LIN {X 0,Y 282.516,Z 713.635,A -85,B 0,C 180,E1 -17402.793,E2 -17402.793} C_VEL
LIN {X 0,Y 282.335,Z 708.345,A -85,B 0,C 180,E1 -17403.944,E2 -17403.944} C_VEL
LIN {X 0,Y 281.852,Z 698.641,A -85,B 0,C 180,E1 -17406.313,E2 -17406.313} C_VEL
LIN {X 0,Y 281.853,Z 692.587,A -85,B 0,C 180,E1 -17407.889,E2 -17407.889} C_VEL
LIN {X 0,Y 281.9,Z 689.303,A -85,B 0,C 180,E1 -17409.389,E2 -17409.389} C_VEL
LIN {X 0,Y 280.609,Z 682.822,A -85,B 0,C 180,E1 -17412.548,E2 -17412.548} C_VEL
LIN {X 0,Y 278.888,Z 673.925,A -85,B 0,C 180,E1 -17417.125,E2 -17417.125} C_VEL
LIN {X 0,Y 277.605,Z 667.473,A -85,B 0,C 180,E1 -17420.734,E2 -17420.734} C_VEL
LIN {X 0,Y 277.296,Z 665.936,A -85,B 0,C 180,E1 -17422.76,E2 -17422.76} C_VEL
LIN {X 0,Y 277.252,Z 665.949,A -85,B 0,C 180,E1 -17426.771,E2 -17426.771} C_VEL
LIN {X 0,Y 277.258,Z 665.946,A -85,B 0,C 180,E1 -17429.538,E2 -17429.538} C_VEL
LIN {X 0,Y 277.355,Z 665.938,A -85,B 0,C 180,E1 -17432.863,E2 -17432.863} C_VEL
LIN {X 0,Y 277.346,Z 666.111,A -85,B 0,C 180,E1 -17435.612,E2 -17435.612} C_VEL
LIN {X 0,Y 278.317,Z 668.775,A -85,B 0,C 180,E1 -17439.297,E2 -17439.297} C_VEL
LIN {X 0,Y 279.682,Z 671.989,A -85,B 0,C 180,E1 -17442.72,E2 -17442.72} C_VEL
LIN {X 0,Y 280.839,Z 675.261,A -85,B 0,C 180,E1 -17445.507,E2 -17445.507} C_VEL
LIN {X 0,Y 282.859,Z 681.56,A -85,B 0,C 180,E1 -17449.984,E2 -17449.984} C_VEL
LIN {X 0,Y 284.181,Z 686.268,A -85,B 0,C 180,E1 -17452.897,E2 -17452.897} C_VEL
LIN {X 0,Y 285.808,Z 694.293,A -85,B 0,C 180,E1 -17457.181,E2 -17457.181} C_VEL
LIN {X 0,Y 286.354,Z 698.631,A -85,B 0,C 180,E1 -17459.297,E2 -17459.297} C_VEL
LIN {X 0,Y 286.469,Z 703.417,A -85,B 0,C 180,E1 -17461.406,E2 -17461.406} C_VEL
LIN {X 0,Y 285.558,Z 710.397,A -85,B 0,C 180,E1 -17464.234,E2 -17464.234} C_VEL
LIN {X 0,Y 283.691,Z 723.175,A -85,B 0,C 180,E1 -17469.266,E2 -17469.266} C_VEL
LIN {X 0,Y 282.575,Z 731.62,A -85,B 0,C 180,E1 -17472.569,E2 -17472.569} C_VEL
LIN {X 0,Y 286.588,Z 745.3,A -85,B 0,C 180,E1 -17473.876,E2 -17473.876} C_VEL
LIN {X 0,Y 288.999,Z 757.39,A -85,B 0,C 180,E1 -17475.109,E2 -17475.109} C_VEL
LIN {X 0,Y 290.187,Z 767.895,A -85,B 0,C 180,E1 -17476.293,E2 -17476.293} C_VEL
LIN {X 0,Y 290.327,Z 771.233,A -85,B 0,C 180,E1 -17476.686,E2 -17476.686} C_VEL
LIN {X 0,Y 288.563,Z 782.164,A -85,B 0,C 180,E1 -17477.917,E2 -17477.917} C_VEL
LIN {X 0,Y 286.272,Z 793.647,A -85,B 0,C 180,E1 -17479.542,E2 -17479.542} C_VEL
LIN {X 0,Y 284.389,Z 802.419,A -85,B 0,C 180,E1 -17481.084,E2 -17481.084} C_VEL
LIN {X 0,Y 282.37,Z 811.035,A -85,B 0,C 180,E1 -17482.945,E2 -17482.945} C_VEL
LIN {X 0,Y 280.37,Z 819.405,A -85,B 0,C 180,E1 -17485.222,E2 -17485.222} C_VEL
LIN {X 0,Y 278.741,Z 825.869,A -85,B 0,C 180,E1 -17487.438,E2 -17487.438} C_VEL
LIN {X 0,Y 277.545,Z 830.747,A -85,B 0,C 180,E1 -17489.571,E2 -17489.571} C_VEL
LIN {X 0,Y 276.408,Z 835.334,A -85,B 0,C 180,E1 -17492.273,E2 -17492.273} C_VEL
LIN {X 0,Y 275.833,Z 837.589,A -85,B 0,C 180,E1 -17494.093,E2 -17494.093} C_VEL
LIN {X 0,Y 275.381,Z 839.172,A -85,B 0,C 180,E1 -17495.943,E2 -17495.943} C_VEL
LIN {X 0,Y 275.105,Z 840.115,A -85,B 0,C 180,E1 -17497.815,E2 -17497.815} C_VEL
LIN {X 0,Y 274.936,Z 840.404,A -85,B 0,C 180,E1 -17499.928,E2 -17499.928} C_VEL
LIN {X 0,Y 274.846,Z 839.806,A -85,B 0,C 180,E1 -17502.138,E2 -17502.138} C_VEL
LIN {X 0,Y 274.987,Z 838.312,A -85,B 0,C 180,E1 -17504.308,E2 -17504.308} C_VEL
LIN {X 0,Y 275.3,Z 835.946,A -85,B 0,C 180,E1 -17506.429,E2 -17506.429} C_VEL
LIN {X 0,Y 275.731,Z 832.732,A -85,B 0,C 180,E1 -17508.495,E2 -17508.495} C_VEL
LIN {X 0,Y 276.231,Z 828.679,A -85,B 0,C 180,E1 -17510.503,E2 -17510.503} C_VEL
LIN {X 0,Y 277.201,Z 822.448,A -85,B 0,C 180,E1 -17512.917,E2 -17512.917} C_VEL
LIN {X 0,Y 278.175,Z 815.947,A -85,B 0,C 180,E1 -17514.911,E2 -17514.911} C_VEL
LIN {X 0,Y 279.558,Z 807.198,A -85,B 0,C 180,E1 -17517.069,E2 -17517.069} C_VEL
LIN {X 0,Y 281.061,Z 797.536,A -85,B 0,C 180,E1 -17518.985,E2 -17518.985} C_VEL
LIN {X 0,Y 282.714,Z 786.024,A -85,B 0,C 180,E1 -17520.79,E2 -17520.79} C_VEL
LIN {X 0,Y 284.124,Z 775.276,A -85,B 0,C 180,E1 -17522.131,E2 -17522.131} C_VEL
LIN {X 0,Y 285.075,Z 766.778,A -85,B 0,C 180,E1 -17522.987,E2 -17522.987} C_VEL
LIN {X 0,Y 283.775,Z 755.666,A -85,B 0,C 180,E1 -17524.046,E2 -17524.046} C_VEL
LIN {X 0,Y 281.716,Z 742.537,A -85,B 0,C 180,E1 -17525.035,E2 -17525.035} C_VEL
LIN {X 0,Y 279.529,Z 730.489,A -85,B 0,C 180,E1 -17525.738,E2 -17525.738} C_VEL
LIN {X 0,Y 280.502,Z 719.526,A -85,B 0,C 180,E1 -17529.849,E2 -17529.849} C_VEL
LIN {X 0,Y 281.518,Z 708.313,A -85,B 0,C 180,E1 -17534.062,E2 -17534.062} C_VEL
LIN {X 0,Y 282.397,Z 698.443,A -85,B 0,C 180,E1 -17537.788,E2 -17537.788} C_VEL
LIN {X 0,Y 282.636,Z 692.781,A -85,B 0,C 180,E1 -17539.977,E2 -17539.977} C_VEL
LIN {X 0,Y 281.744,Z 685.786,A -85,B 0,C 180,E1 -17542.836,E2 -17542.836} C_VEL
LIN {X 0,Y 280.07,Z 677.374,A -85,B 0,C 180,E1 -17546.404,E2 -17546.404} C_VEL
LIN {X 0,Y 278.607,Z 668.999,A -85,B 0,C 180,E1 -17550.001,E2 -17550.001} C_VEL
LIN {X 0,Y 277.825,Z 665.875,A -85,B 0,C 180,E1 -17551.45,E2 -17551.45} C_VEL
LIN {X 0,Y 277.651,Z 665.897,A -85,B 0,C 180,E1 -17557.272,E2 -17557.272} C_VEL
LIN {X 0,Y 277.508,Z 665.911,A -85,B 0,C 180,E1 -17560.212,E2 -17560.212} C_VEL
LIN {X 0,Y 277.436,Z 665.927,A -85,B 0,C 180,E1 -17564.16,E2 -17564.16} C_VEL
LIN {X 0,Y 281.89,Z 679.397,A -85,B 0,C 180,E1 -17565.735,E2 -17565.735} C_VEL
LIN {X 0,Y 284.669,Z 688.988,A -85,B 0,C 180,E1 -17567.051,E2 -17567.051} C_VEL
LIN {X 0,Y 285.979,Z 694.54,A -85,B 0,C 180,E1 -17567.891,E2 -17567.891} C_VEL
LIN {X 0,Y 284.721,Z 705.21,A -85,B 0,C 180,E1 -17569.466,E2 -17569.466} C_VEL
LIN {X 0,Y 283.372,Z 715.102,A -85,B 0,C 180,E1 -17571.268,E2 -17571.268} C_VEL
LIN {X 0,Y 282.092,Z 723.419,A -85,B 0,C 180,E1 -17573.126,E2 -17573.126} C_VEL
LIN {X 0,Y 280.89,Z 730.843,A -85,B 0,C 180,E1 -17575.173,E2 -17575.173} C_VEL
LIN {X 0,Y 279.764,Z 737.817,A -85,B 0,C 180,E1 -17577.59,E2 -17577.59} C_VEL
LIN {X 0,Y 278.868,Z 743.707,A -85,B 0,C 180,E1 -17580.268,E2 -17580.268} C_VEL
LIN {X 0,Y 278.373,Z 746.65,A -85,B 0,C 180,E1 -17582.018,E2 -17582.018} C_VEL
LIN {X 0,Y 278.006,Z 748.956,A -85,B 0,C 180,E1 -17583.791,E2 -17583.791} C_VEL
LIN {X 0,Y 277.752,Z 750.928,A -85,B 0,C 180,E1 -17585.934,E2 -17585.934} C_VEL
LIN {X 0,Y 277.767,Z 752.085,A -85,B 0,C 180,E1 -17588.339,E2 -17588.339} C_VEL
LIN {X 0,Y 278.168,Z 752.088,A -85,B 0,C 180,E1 -17591.064,E2 -17591.064} C_VEL
LIN {X 0,Y 278.594,Z 751.262,A -85,B 0,C 180,E1 -17592.982,E2 -17592.982} C_VEL
LIN {X 0,Y 279.307,Z 749.426,A -85,B 0,C 180,E1 -17595.207,E2 -17595.207} C_VEL
LIN {X 0,Y 280.569,Z 745.778,A -85,B 0,C 180,E1 -17597.935,E2 -17597.935} C_VEL
LIN {X 0,Y 282.038,Z 740.635,A -85,B 0,C 180,E1 -17600.578,E2 -17600.578} C_VEL
LIN {X 0,Y 283.861,Z 734.085,A -85,B 0,C 180,E1 -17603.052,E2 -17603.052} C_VEL
LIN {X 0,Y 285.785,Z 726.31,A -85,B 0,C 180,E1 -17605.317,E2 -17605.317} C_VEL
LIN {X 0,Y 287.637,Z 717.926,A -85,B 0,C 180,E1 -17607.249,E2 -17607.249} C_VEL
LIN {X 0,Y 289.479,Z 709.01,A -85,B 0,C 180,E1 -17608.9,E2 -17608.9} C_VEL
LIN {X 0,Y 290.619,Z 701.513,A -85,B 0,C 180,E1 -17610.082,E2 -17610.082} C_VEL
LIN {X 0,Y 288.425,Z 693.11,A -85,B 0,C 180,E1 -17611.631,E2 -17611.631} C_VEL
LIN {X 0,Y 285.145,Z 683.447,A -85,B 0,C 180,E1 -17613.269,E2 -17613.269} C_VEL
LIN {X 0,Y 280.932,Z 673.769,A -85,B 0,C 180,E1 -17614.832,E2 -17614.832} C_VEL
LIN {X 0,Y 278.336,Z 668.845,A -85,B 0,C 180,E1 -17615.621,E2 -17615.621} C_VEL
LIN {X 0,Y 277.301,Z 665.938,A -85,B 0,C 180,E1 -17616,E2 -17616} C_VEL
LIN {X 0,Y 277.347,Z 665.939,A -85,B 0,C 180,E1 -17620.767,E2 -17620.767} C_VEL
LIN {X 0,Y 277.437,Z 665.925,A -85,B 0,C 180,E1 -17625.326,E2 -17625.326} C_VEL
LIN {X 0,Y 277.406,Z 665.927,A -85,B 0,C 180,E1 -17625.963,E2 -17625.963} C_VEL
LIN {X 0,Y 276.737,Z 666.015,A -85,B 0,C 180,E1 -17627.175,E2 -17627.175} C_VEL
LIN {X 0,Y 273.935,Z 666.357,A -85,B 0,C 180,E1 -17629.153,E2 -17629.153} C_VEL
LIN {X 0,Y 271.603,Z 666.652,A -85,B 0,C 180,E1 -17630.761,E2 -17630.761} C_VEL
LIN {X 0,Y 270.654,Z 666.761,A -85,B 0,C 180,E1 -17632.004,E2 -17632.004} C_VEL
LIN {X 0,Y 270.604,Z 666.766,A -85,B 0,C 180,E1 -17632.425,E2 -17632.425} C_VEL
LIN {X 0,Y 270.79,Z 666.754,A -85,B 0,C 180,E1 -17638.513,E2 -17638.513} C_VEL
LIN {X 0,Y 270.79,Z 666.742,A -85,B 0,C 180,E1 -17641.487,E2 -17641.487} C_VEL
LIN {X 0,Y 270.614,Z 666.776,A -85,B 0,C 180,E1 -17647.461,E2 -17647.461} C_VEL
LIN {X 0,Y 270.444,Z 666.795,A -85,B 0,C 180,E1 -17650.481,E2 -17650.481} C_VEL
LIN {X 0,Y 270.406,Z 666.802,A -85,B 0,C 180,E1 -17655.065,E2 -17655.065} C_VEL
LIN {X 0,Y 270.304,Z 666.807,A -85,B 0,C 180,E1 -17659.756,E2 -17659.756} C_VEL
LIN {X 0,Y 270.276,Z 666.819,A -85,B 0,C 180,E1 -17664.586,E2 -17664.586} C_VEL
LIN {X 0,Y 270.272,Z 666.816,A -85,B 0,C 180,E1 -17667.909,E2 -17667.909} C_VEL
LIN {X 0,Y 270.187,Z 666.83,A -85,B 0,C 180,E1 -17671.348,E2 -17671.348} C_VEL
LIN {X 0,Y 270.224,Z 666.943,A -85,B 0,C 180,E1 -17673.529,E2 -17673.529} C_VEL
LIN {X 0,Y 271.355,Z 671.877,A -85,B 0,C 180,E1 -17677.492,E2 -17677.492} C_VEL
LIN {X 0,Y 272.72,Z 678.439,A -85,B 0,C 180,E1 -17682.069,E2 -17682.069} C_VEL
LIN {X 0,Y 273.966,Z 685.04,A -85,B 0,C 180,E1 -17686.161,E2 -17686.161} C_VEL
LIN {X 0,Y 275.274,Z 692.519,A -85,B 0,C 180,E1 -17690.336,E2 -17690.336} C_VEL
LIN {X 0,Y 275.316,Z 694.363,A -85,B 0,C 180,E1 -17691.287,E2 -17691.287} C_VEL
LIN {X 0,Y 273.666,Z 702.79,A -85,B 0,C 180,E1 -17695.265,E2 -17695.265} C_VEL
LIN {X 0,Y 271.808,Z 713.574,A -85,B 0,C 180,E1 -17700.149,E2 -17700.149} C_VEL
LIN {X 0,Y 271.718,Z 714.564,A -85,B 0,C 180,E1 -17700.511,E2 -17700.511} C_VEL
LIN {X 0,Y 274.842,Z 729.066,A -85,B 0,C 180,E1 -17701.706,E2 -17701.706} C_VEL
LIN {X 0,Y 276.656,Z 742.403,A -85,B 0,C 180,E1 -17702.962,E2 -17702.962} C_VEL
LIN {X 0,Y 277.427,Z 754.489,A -85,B 0,C 180,E1 -17704.276,E2 -17704.276} C_VEL
LIN {X 0,Y 277.294,Z 766.965,A -85,B 0,C 180,E1 -17705.842,E2 -17705.842} C_VEL
LIN {X 0,Y 276.639,Z 775.939,A -85,B 0,C 180,E1 -17707.11,E2 -17707.11} C_VEL
LIN {X 0,Y 276.576,Z 788.697,A -85,B 0,C 180,E1 -17708.379,E2 -17708.379} C_VEL
LIN {X 0,Y 275.815,Z 796.463,A -85,B 0,C 180,E1 -17709.295,E2 -17709.295} C_VEL
LIN {X 0,Y 274.239,Z 806.674,A -85,B 0,C 180,E1 -17710.734,E2 -17710.734} C_VEL
LIN {X 0,Y 272.809,Z 816.634,A -85,B 0,C 180,E1 -17712.483,E2 -17712.483} C_VEL
LIN {X 0,Y 271.598,Z 824.755,A -85,B 0,C 180,E1 -17714.234,E2 -17714.234} C_VEL
LIN {X 0,Y 270.302,Z 833.109,A -85,B 0,C 180,E1 -17716.466,E2 -17716.466} C_VEL
LIN {X 0,Y 269.369,Z 839.817,A -85,B 0,C 180,E1 -17718.715,E2 -17718.715} C_VEL
LIN {X 0,Y 268.762,Z 845.144,A -85,B 0,C 180,E1 -17720.972,E2 -17720.972} C_VEL
LIN {X 0,Y 268.426,Z 849.255,A -85,B 0,C 180,E1 -17723.233,E2 -17723.233} C_VEL
LIN {X 0,Y 268.262,Z 852.262,A -85,B 0,C 180,E1 -17725.491,E2 -17725.491} C_VEL
LIN {X 0,Y 268.275,Z 853.702,A -85,B 0,C 180,E1 -17726.996,E2 -17726.996} C_VEL
LIN {X 0,Y 268.277,Z 854.694,A -85,B 0,C 180,E1 -17728.498,E2 -17728.498} C_VEL
LIN {X 0,Y 268.298,Z 855.284,A -85,B 0,C 180,E1 -17729.999,E2 -17729.999} C_VEL
LIN {X 0,Y 268.265,Z 855.467,A -85,B 0,C 180,E1 -17731.5,E2 -17731.5} C_VEL
LIN {X 0,Y 268.247,Z 855.199,A -85,B 0,C 180,E1 -17733.003,E2 -17733.003} C_VEL
LIN {X 0,Y 268.31,Z 853.465,A -85,B 0,C 180,E1 -17736.013,E2 -17736.013} C_VEL
LIN {X 0,Y 268.52,Z 851.985,A -85,B 0,C 180,E1 -17737.519,E2 -17737.519} C_VEL
LIN {X 0,Y 269.047,Z 848.948,A -85,B 0,C 180,E1 -17739.775,E2 -17739.775} C_VEL
LIN {X 0,Y 269.882,Z 844.869,A -85,B 0,C 180,E1 -17742.023,E2 -17742.023} C_VEL
LIN {X 0,Y 271.316,Z 838.624,A -85,B 0,C 180,E1 -17744.628,E2 -17744.628} C_VEL
LIN {X 0,Y 273.088,Z 831.856,A -85,B 0,C 180,E1 -17746.828,E2 -17746.828} C_VEL
LIN {X 0,Y 274.777,Z 824.228,A -85,B 0,C 180,E1 -17748.851,E2 -17748.851} C_VEL
LIN {X 0,Y 276.976,Z 815.012,A -85,B 0,C 180,E1 -17750.807,E2 -17750.807} C_VEL
LIN {X 0,Y 279.372,Z 804.653,A -85,B 0,C 180,E1 -17752.558,E2 -17752.558} C_VEL
LIN {X 0,Y 281.353,Z 794.523,A -85,B 0,C 180,E1 -17753.947,E2 -17753.947} C_VEL
LIN {X 0,Y 282.205,Z 783.816,A -85,B 0,C 180,E1 -17755.237,E2 -17755.237} C_VEL
LIN {X 0,Y 282.791,Z 772.129,A -85,B 0,C 180,E1 -17756.367,E2 -17756.367} C_VEL
LIN {X 0,Y 282.217,Z 761.442,A -85,B 0,C 180,E1 -17757.306,E2 -17757.306} C_VEL
LIN {X 0,Y 280.394,Z 749.6,A -85,B 0,C 180,E1 -17758.265,E2 -17758.265} C_VEL
LIN {X 0,Y 277.549,Z 737.167,A -85,B 0,C 180,E1 -17759.29,E2 -17759.29} C_VEL
LIN {X 0,Y 276.992,Z 723.016,A -85,B 0,C 180,E1 -17761.98,E2 -17761.98} C_VEL
LIN {X 0,Y 276.498,Z 710.459,A -85,B 0,C 180,E1 -17764.762,E2 -17764.762} C_VEL
LIN {X 0,Y 276.237,Z 700.914,A -85,B 0,C 180,E1 -17767.173,E2 -17767.173} C_VEL
LIN {X 0,Y 276.348,Z 695.937,A -85,B 0,C 180,E1 -17768.539,E2 -17768.539} C_VEL
LIN {X 0,Y 275.257,Z 690.441,A -85,B 0,C 180,E1 -17770.572,E2 -17770.572} C_VEL
LIN {X 0,Y 273.681,Z 683.277,A -85,B 0,C 180,E1 -17773.894,E2 -17773.894} C_VEL
LIN {X 0,Y 272.784,Z 677.893,A -85,B 0,C 180,E1 -17776.941,E2 -17776.941} C_VEL
LIN {X 0,Y 272.529,Z 672.615,A -85,B 0,C 180,E1 -17780.68,E2 -17780.68} C_VEL
LIN {X 0,Y 272.368,Z 671.627,A -85,B 0,C 180,E1 -17781.736,E2 -17781.736} C_VEL
LIN {X 0,Y 271.899,Z 670.538,A -85,B 0,C 180,E1 -17783.523,E2 -17783.523} C_VEL
LIN {X 0,Y 271.093,Z 669.499,A -85,B 0,C 180,E1 -17787.015,E2 -17787.015} C_VEL
LIN {X 0,Y 271.016,Z 669.352,A -85,B 0,C 180,E1 -17790.481,E2 -17790.481} C_VEL
LIN {X 0,Y 271.763,Z 670.36,A -85,B 0,C 180,E1 -17794.837,E2 -17794.837} C_VEL
LIN {X 0,Y 272.599,Z 672.91,A -85,B 0,C 180,E1 -17798.842,E2 -17798.842} C_VEL
LIN {X 0,Y 273.689,Z 675.62,A -85,B 0,C 180,E1 -17802.052,E2 -17802.052} C_VEL
LIN {X 0,Y 275.21,Z 680.045,A -85,B 0,C 180,E1 -17806.02,E2 -17806.02} C_VEL
LIN {X 0,Y 276.81,Z 685.119,A -85,B 0,C 180,E1 -17809.762,E2 -17809.762} C_VEL
LIN {X 0,Y 278.052,Z 689.768,A -85,B 0,C 180,E1 -17812.739,E2 -17812.739} C_VEL
LIN {X 0,Y 279.519,Z 697.573,A -85,B 0,C 180,E1 -17817.117,E2 -17817.117} C_VEL
LIN {X 0,Y 280.009,Z 702.002,A -85,B 0,C 180,E1 -17819.281,E2 -17819.281} C_VEL
LIN {X 0,Y 279.929,Z 706.769,A -85,B 0,C 180,E1 -17821.438,E2 -17821.438} C_VEL
LIN {X 0,Y 278.841,Z 713.804,A -85,B 0,C 180,E1 -17824.336,E2 -17824.336} C_VEL
LIN {X 0,Y 277.155,Z 724.731,A -85,B 0,C 180,E1 -17828.751,E2 -17828.751} C_VEL
LIN {X 0,Y 276.136,Z 731.883,A -85,B 0,C 180,E1 -17831.608,E2 -17831.608} C_VEL
LIN {X 0,Y 280.408,Z 746.094,A -85,B 0,C 180,E1 -17833.036,E2 -17833.036} C_VEL
LIN {X 0,Y 282.806,Z 758.54,A -85,B 0,C 180,E1 -17834.389,E2 -17834.389} C_VEL
LIN {X 0,Y 284,Z 770.352,A -85,B 0,C 180,E1 -17835.796,E2 -17835.796} C_VEL
LIN {X 0,Y 283.702,Z 775.24,A -85,B 0,C 180,E1 -17836.367,E2 -17836.367} C_VEL
LIN {X 0,Y 281.675,Z 785.865,A -85,B 0,C 180,E1 -17837.659,E2 -17837.659} C_VEL
LIN {X 0,Y 279.455,Z 796.319,A -85,B 0,C 180,E1 -17839.273,E2 -17839.273} C_VEL
LIN {X 0,Y 277.085,Z 806.254,A -85,B 0,C 180,E1 -17841.188,E2 -17841.188} C_VEL
LIN {X 0,Y 275.074,Z 814.242,A -85,B 0,C 180,E1 -17843.109,E2 -17843.109} C_VEL
LIN {X 0,Y 273.2,Z 821.576,A -85,B 0,C 180,E1 -17845.31,E2 -17845.31} C_VEL
LIN {X 0,Y 271.388,Z 828.098,A -85,B 0,C 180,E1 -17847.784,E2 -17847.784} C_VEL
LIN {X 0,Y 270.164,Z 832.914,A -85,B 0,C 180,E1 -17850.18,E2 -17850.18} C_VEL
LIN {X 0,Y 269.297,Z 836.161,A -85,B 0,C 180,E1 -17852.344,E2 -17852.344} C_VEL
LIN {X 0,Y 268.466,Z 839.02,A -85,B 0,C 180,E1 -17855.164,E2 -17855.164} C_VEL
LIN {X 0,Y 267.967,Z 840.473,A -85,B 0,C 180,E1 -17858.113,E2 -17858.113} C_VEL
LIN {X 0,Y 267.783,Z 840.39,A -85,B 0,C 180,E1 -17861.005,E2 -17861.005} C_VEL
LIN {X 0,Y 267.795,Z 839.456,A -85,B 0,C 180,E1 -17863.027,E2 -17863.027} C_VEL
LIN {X 0,Y 268.136,Z 836.58,A -85,B 0,C 180,E1 -17866.077,E2 -17866.077} C_VEL
LIN {X 0,Y 268.571,Z 833.554,A -85,B 0,C 180,E1 -17868.182,E2 -17868.182} C_VEL
LIN {X 0,Y 269.219,Z 828.568,A -85,B 0,C 180,E1 -17870.756,E2 -17870.756} C_VEL
LIN {X 0,Y 270.232,Z 822.128,A -85,B 0,C 180,E1 -17873.263,E2 -17873.263} C_VEL
LIN {X 0,Y 271.452,Z 814.368,A -85,B 0,C 180,E1 -17875.622,E2 -17875.622} C_VEL
LIN {X 0,Y 272.882,Z 805.731,A -85,B 0,C 180,E1 -17877.718,E2 -17877.718} C_VEL
LIN {X 0,Y 274.556,Z 795.036,A -85,B 0,C 180,E1 -17879.778,E2 -17879.778} C_VEL
LIN {X 0,Y 276.174,Z 784.204,A -85,B 0,C 180,E1 -17881.437,E2 -17881.437} C_VEL
LIN {X 0,Y 277.521,Z 773.78,A -85,B 0,C 180,E1 -17882.71,E2 -17882.71} C_VEL
LIN {X 0,Y 278.159,Z 766.612,A -85,B 0,C 180,E1 -17883.45,E2 -17883.45} C_VEL
LIN {X 0,Y 276.72,Z 754.813,A -85,B 0,C 180,E1 -17884.596,E2 -17884.596} C_VEL
LIN {X 0,Y 274.596,Z 741.045,A -85,B 0,C 180,E1 -17885.63,E2 -17885.63} C_VEL
LIN {X 0,Y 272.611,Z 730.637,A -85,B 0,C 180,E1 -17886.247,E2 -17886.247} C_VEL
LIN {X 0,Y 273.6,Z 720.504,A -85,B 0,C 180,E1 -17890.103,E2 -17890.103} C_VEL
LIN {X 0,Y 274.655,Z 709.243,A -85,B 0,C 180,E1 -17894.415,E2 -17894.415} C_VEL
LIN {X 0,Y 275.579,Z 699.289,A -85,B 0,C 180,E1 -17898.229,E2 -17898.229} C_VEL
LIN {X 0,Y 275.72,Z 693.635,A -85,B 0,C 180,E1 -17900.464,E2 -17900.464} C_VEL
LIN {X 0,Y 274.774,Z 686.612,A -85,B 0,C 180,E1 -17903.392,E2 -17903.392} C_VEL
LIN {X 0,Y 272.555,Z 674.785,A -85,B 0,C 180,E1 -17908.523,E2 -17908.523} C_VEL
LIN {X 0,Y 271.508,Z 669.803,A -85,B 0,C 180,E1 -17910.742,E2 -17910.742} C_VEL
LIN {X 0,Y 270.71,Z 666.763,A -85,B 0,C 180,E1 -17912.233,E2 -17912.233} C_VEL
LIN {X 0,Y 270.609,Z 666.775,A -85,B 0,C 180,E1 -17917.462,E2 -17917.462} C_VEL
LIN {X 0,Y 270.443,Z 666.793,A -85,B 0,C 180,E1 -17920.482,E2 -17920.482} C_VEL
LIN {X 0,Y 270.406,Z 666.804,A -85,B 0,C 180,E1 -17923.624,E2 -17923.624} C_VEL
LIN {X 0,Y 274.776,Z 679.978,A -85,B 0,C 180,E1 -17925.199,E2 -17925.199} C_VEL
LIN {X 0,Y 277.625,Z 689.557,A -85,B 0,C 180,E1 -17926.547,E2 -17926.547} C_VEL
LIN {X 0,Y 279.157,Z 696.219,A -85,B 0,C 180,E1 -17927.585,E2 -17927.585} C_VEL
LIN {X 0,Y 277.848,Z 706.788,A -85,B 0,C 180,E1 -17929.198,E2 -17929.198} C_VEL
LIN {X 0,Y 276.591,Z 715.581,A -85,B 0,C 180,E1 -17930.839,E2 -17930.839} C_VEL
LIN {X 0,Y 275.239,Z 724.199,A -85,B 0,C 180,E1 -17932.793,E2 -17932.793} C_VEL
LIN {X 0,Y 273.897,Z 732.171,A -85,B 0,C 180,E1 -17935.049,E2 -17935.049} C_VEL
LIN {X 0,Y 272.715,Z 739.374,A -85,B 0,C 180,E1 -17937.638,E2 -17937.638} C_VEL
LIN {X 0,Y 271.841,Z 744.913,A -85,B 0,C 180,E1 -17940.275,E2 -17940.275} C_VEL
LIN {X 0,Y 271.139,Z 749.043,A -85,B 0,C 180,E1 -17942.979,E2 -17942.979} C_VEL
LIN {X 0,Y 270.837,Z 751.025,A -85,B 0,C 180,E1 -17944.812,E2 -17944.812} C_VEL
LIN {X 0,Y 270.721,Z 752.399,A -85,B 0,C 180,E1 -17946.662,E2 -17946.662} C_VEL
LIN {X 0,Y 270.799,Z 753.217,A -85,B 0,C 180,E1 -17948.869,E2 -17948.869} C_VEL
LIN {X 0,Y 271.185,Z 753.134,A -85,B 0,C 180,E1 -17951.275,E2 -17951.275} C_VEL
LIN {X 0,Y 271.982,Z 751.621,A -85,B 0,C 180,E1 -17954.242,E2 -17954.242} C_VEL
LIN {X 0,Y 273.179,Z 748.538,A -85,B 0,C 180,E1 -17957.143,E2 -17957.143} C_VEL
LIN {X 0,Y 274.2,Z 745.441,A -85,B 0,C 180,E1 -17959.123,E2 -17959.123} C_VEL
LIN {X 0,Y 275.78,Z 740.327,A -85,B 0,C 180,E1 -17961.595,E2 -17961.595} C_VEL
LIN {X 0,Y 277.297,Z 734.91,A -85,B 0,C 180,E1 -17963.62,E2 -17963.62} C_VEL
LIN {X 0,Y 279.062,Z 728.248,A -85,B 0,C 180,E1 -17965.625,E2 -17965.625} C_VEL
LIN {X 0,Y 281.006,Z 719.94,A -85,B 0,C 180,E1 -17967.633,E2 -17967.633} C_VEL
LIN {X 0,Y 283.014,Z 710.786,A -85,B 0,C 180,E1 -17969.399,E2 -17969.399} C_VEL
LIN {X 0,Y 284.218,Z 703.649,A -85,B 0,C 180,E1 -17970.569,E2 -17970.569} C_VEL
LIN {X 0,Y 282.124,Z 695.459,A -85,B 0,C 180,E1 -17972.155,E2 -17972.155} C_VEL
LIN {X 0,Y 278.989,Z 686.089,A -85,B 0,C 180,E1 -17973.843,E2 -17973.843} C_VEL
LIN {X 0,Y 274.729,Z 676.384,A -85,B 0,C 180,E1 -17975.522,E2 -17975.522} C_VEL
LIN {X 0,Y 271.46,Z 669.995,A -85,B 0,C 180,E1 -17976.594,E2 -17976.594} C_VEL
LIN {X 0,Y 270.292,Z 667.295,A -85,B 0,C 180,E1 -17976.994,E2 -17976.994} C_VEL
LIN {X 0,Y 270.234,Z 666.811,A -85,B 0,C 180,E1 -17977.09,E2 -17977.09} C_VEL
LIN {X 0,Y 270.303,Z 666.816,A -85,B 0,C 180,E1 -17980.245,E2 -17980.245} C_VEL
LIN {X 0,Y 270.405,Z 666.804,A -85,B 0,C 180,E1 -17984.936,E2 -17984.936} C_VEL
LIN {X 0,Y 270.444,Z 666.793,A -85,B 0,C 180,E1 -17989.519,E2 -17989.519} C_VEL
LIN {X 0,Y 270.604,Z 666.766,A -85,B 0,C 180,E1 -17992.425,E2 -17992.425} C_VEL
LIN {X 0,Y 270.018,Z 666.846,A -85,B 0,C 180,E1 -17993.666,E2 -17993.666} C_VEL
LIN {X 0,Y 267.236,Z 667.195,A -85,B 0,C 180,E1 -17995.69,E2 -17995.69} C_VEL
LIN {X 0,Y 264.841,Z 667.496,A -85,B 0,C 180,E1 -17997.335,E2 -17997.335} C_VEL
LIN {X 0,Y 263.825,Z 667.621,A -85,B 0,C 180,E1 -17998.61,E2 -17998.61} C_VEL
LIN {X 0,Y 263.751,Z 667.625,A -85,B 0,C 180,E1 -17999.041,E2 -17999.041} C_VEL
LIN {X 0,Y 263.754,Z 667.619,A -85,B 0,C 180,E1 -18001.527,E2 -18001.527} C_VEL
LIN {X 0,Y 263.575,Z 667.652,A -85,B 0,C 180,E1 -18007.662,E2 -18007.662} C_VEL
LIN {X 0,Y 263.377,Z 667.679,A -85,B 0,C 180,E1 -18010.766,E2 -18010.766} C_VEL
LIN {X 0,Y 263.354,Z 667.679,A -85,B 0,C 180,E1 -18015.478,E2 -18015.478} C_VEL
LIN {X 0,Y 263.266,Z 667.684,A -85,B 0,C 180,E1 -18020.307,E2 -18020.307} C_VEL
LIN {X 0,Y 263.21,Z 667.695,A -85,B 0,C 180,E1 -18025.291,E2 -18025.291} C_VEL
LIN {X 0,Y 263.178,Z 667.7,A -85,B 0,C 180,E1 -18028.73,E2 -18028.73} C_VEL
LIN {X 0,Y 263.135,Z 667.799,A -85,B 0,C 180,E1 -18032.288,E2 -18032.288} C_VEL
LIN {X 0,Y 264.117,Z 671.885,A -85,B 0,C 180,E1 -18035.832,E2 -18035.832} C_VEL
LIN {X 0,Y 265.195,Z 677.091,A -85,B 0,C 180,E1 -18039.777,E2 -18039.777} C_VEL
LIN {X 0,Y 266.263,Z 682.303,A -85,B 0,C 180,E1 -18043.336,E2 -18043.336} C_VEL
LIN {X 0,Y 267.445,Z 688.889,A -85,B 0,C 180,E1 -18047.375,E2 -18047.375} C_VEL
LIN {X 0,Y 268.347,Z 694.049,A -85,B 0,C 180,E1 -18050.288,E2 -18050.288} C_VEL
LIN {X 0,Y 268.092,Z 697.076,A -85,B 0,C 180,E1 -18051.855,E2 -18051.855} C_VEL
LIN {X 0,Y 266.473,Z 704.694,A -85,B 0,C 180,E1 -18055.527,E2 -18055.527} C_VEL
LIN {X 0,Y 264.967,Z 713.004,A -85,B 0,C 180,E1 -18059.407,E2 -18059.407} C_VEL
LIN {X 0,Y 265.915,Z 717.051,A -85,B 0,C 180,E1 -18059.759,E2 -18059.759} C_VEL
LIN {X 0,Y 268.598,Z 730.061,A -85,B 0,C 180,E1 -18060.947,E2 -18060.947} C_VEL
LIN {X 0,Y 270.275,Z 743.125,A -85,B 0,C 180,E1 -18062.272,E2 -18062.272} C_VEL
LIN {X 0,Y 270.94,Z 754.77,A -85,B 0,C 180,E1 -18063.615,E2 -18063.615} C_VEL
LIN {X 0,Y 270.739,Z 766.246,A -85,B 0,C 180,E1 -18065.127,E2 -18065.127} C_VEL
LIN {X 0,Y 269.781,Z 777.533,A -85,B 0,C 180,E1 -18066.811,E2 -18066.811} C_VEL
LIN {X 0,Y 269.708,Z 788.94,A -85,B 0,C 180,E1 -18068.001,E2 -18068.001} C_VEL
LIN {X 0,Y 268.936,Z 796.627,A -85,B 0,C 180,E1 -18068.941,E2 -18068.941} C_VEL
LIN {X 0,Y 267.319,Z 806.772,A -85,B 0,C 180,E1 -18070.414,E2 -18070.414} C_VEL
LIN {X 0,Y 265.833,Z 816.802,A -85,B 0,C 180,E1 -18072.232,E2 -18072.232} C_VEL
LIN {X 0,Y 264.453,Z 825.502,A -85,B 0,C 180,E1 -18074.192,E2 -18074.192} C_VEL
LIN {X 0,Y 263.145,Z 833.683,A -85,B 0,C 180,E1 -18076.485,E2 -18076.485} C_VEL
LIN {X 0,Y 262.364,Z 839.241,A -85,B 0,C 180,E1 -18078.409,E2 -18078.409} C_VEL
LIN {X 0,Y 261.726,Z 844.645,A -85,B 0,C 180,E1 -18080.728,E2 -18080.728} C_VEL
LIN {X 0,Y 261.353,Z 848.825,A -85,B 0,C 180,E1 -18083.049,E2 -18083.049} C_VEL
LIN {X 0,Y 261.18,Z 851.897,A -85,B 0,C 180,E1 -18085.369,E2 -18085.369} C_VEL
LIN {X 0,Y 261.185,Z 853.396,A -85,B 0,C 180,E1 -18086.914,E2 -18086.914} C_VEL
LIN {X 0,Y 261.201,Z 854.42,A -85,B 0,C 180,E1 -18088.457,E2 -18088.457} C_VEL
LIN {X 0,Y 261.22,Z 855.038,A -85,B 0,C 180,E1 -18089.999,E2 -18089.999} C_VEL
LIN {X 0,Y 261.19,Z 855.255,A -85,B 0,C 180,E1 -18091.541,E2 -18091.541} C_VEL
LIN {X 0,Y 261.158,Z 855.04,A -85,B 0,C 180,E1 -18093.084,E2 -18093.084} C_VEL
LIN {X 0,Y 261.237,Z 853.374,A -85,B 0,C 180,E1 -18096.177,E2 -18096.177} C_VEL
LIN {X 0,Y 261.449,Z 851.948,A -85,B 0,C 180,E1 -18097.723,E2 -18097.723} C_VEL
LIN {X 0,Y 262.034,Z 848.97,A -85,B 0,C 180,E1 -18100.039,E2 -18100.039} C_VEL
LIN {X 0,Y 262.92,Z 844.964,A -85,B 0,C 180,E1 -18102.347,E2 -18102.347} C_VEL
LIN {X 0,Y 264.161,Z 839.821,A -85,B 0,C 180,E1 -18104.639,E2 -18104.639} C_VEL
LIN {X 0,Y 265.991,Z 833.393,A -85,B 0,C 180,E1 -18106.895,E2 -18106.895} C_VEL
LIN {X 0,Y 267.949,Z 825.162,A -85,B 0,C 180,E1 -18109.223,E2 -18109.223} C_VEL
LIN {X 0,Y 270.399,Z 815.678,A -85,B 0,C 180,E1 -18111.337,E2 -18111.337} C_VEL
LIN {X 0,Y 272.886,Z 805.489,A -85,B 0,C 180,E1 -18113.125,E2 -18113.125} C_VEL
LIN {X 0,Y 274.957,Z 795.57,A -85,B 0,C 180,E1 -18114.541,E2 -18114.541} C_VEL
LIN {X 0,Y 275.959,Z 785.051,A -85,B 0,C 180,E1 -18115.875,E2 -18115.875} C_VEL
LIN {X 0,Y 276.717,Z 774.001,A -85,B 0,C 180,E1 -18117.018,E2 -18117.018} C_VEL
LIN {X 0,Y 276.373,Z 763.886,A -85,B 0,C 180,E1 -18117.964,E2 -18117.964} C_VEL
LIN {X 0,Y 274.755,Z 752.009,A -85,B 0,C 180,E1 -18118.997,E2 -18118.997} C_VEL
LIN {X 0,Y 271.405,Z 737.257,A -85,B 0,C 180,E1 -18120.273,E2 -18120.273} C_VEL
LIN {X 0,Y 271.013,Z 723.771,A -85,B 0,C 180,E1 -18122.995,E2 -18122.995} C_VEL
LIN {X 0,Y 270.813,Z 714.062,A -85,B 0,C 180,E1 -18125.228,E2 -18125.228} C_VEL
LIN {X 0,Y 270.671,Z 704.472,A -85,B 0,C 180,E1 -18127.715,E2 -18127.715} C_VEL
LIN {X 0,Y 270.919,Z 700.327,A -85,B 0,C 180,E1 -18128.9,E2 -18128.9} C_VEL
LIN {X 0,Y 270.119,Z 695.671,A -85,B 0,C 180,E1 -18130.574,E2 -18130.574} C_VEL
LIN {X 0,Y 268.642,Z 688.778,A -85,B 0,C 180,E1 -18133.741,E2 -18133.741} C_VEL
LIN {X 0,Y 267.652,Z 683.02,A -85,B 0,C 180,E1 -18136.944,E2 -18136.944} C_VEL
LIN {X 0,Y 267.453,Z 677.449,A -85,B 0,C 180,E1 -18140.901,E2 -18140.901} C_VEL
LIN {X 0,Y 267.036,Z 675.931,A -85,B 0,C 180,E1 -18142.747,E2 -18142.747} C_VEL
LIN {X 0,Y 266.047,Z 674.533,A -85,B 0,C 180,E1 -18146.307,E2 -18146.307} C_VEL
LIN {X 0,Y 265.77,Z 674.123,A -85,B 0,C 180,E1 -18150.765,E2 -18150.765} C_VEL
LIN {X 0,Y 266.4,Z 675.06,A -85,B 0,C 180,E1 -18155.032,E2 -18155.032} C_VEL
LIN {X 0,Y 267.398,Z 678.216,A -85,B 0,C 180,E1 -18160.021,E2 -18160.021} C_VEL
LIN {X 0,Y 268.435,Z 681.088,A -85,B 0,C 180,E1 -18163.262,E2 -18163.262} C_VEL
LIN {X 0,Y 269.538,Z 684.62,A -85,B 0,C 180,E1 -18166.428,E2 -18166.428} C_VEL
LIN {X 0,Y 271.043,Z 689.584,A -85,B 0,C 180,E1 -18170.162,E2 -18170.162} C_VEL
LIN {X 0,Y 271.909,Z 693.229,A -85,B 0,C 180,E1 -18172.574,E2 -18172.574} C_VEL
LIN {X 0,Y 273.299,Z 701.024,A -85,B 0,C 180,E1 -18177.052,E2 -18177.052} C_VEL
LIN {X 0,Y 273.697,Z 706.906,A -85,B 0,C 180,E1 -18180,E2 -18180} C_VEL
LIN {X 0,Y 273.151,Z 711.922,A -85,B 0,C 180,E1 -18182.212,E2 -18182.212} C_VEL
LIN {X 0,Y 271.237,Z 722.701,A -85,B 0,C 180,E1 -18186.696,E2 -18186.696} C_VEL
LIN {X 0,Y 269.806,Z 732.132,A -85,B 0,C 180,E1 -18190.553,E2 -18190.553} C_VEL
LIN {X 0,Y 273.847,Z 745.446,A -85,B 0,C 180,E1 -18191.988,E2 -18191.988} C_VEL
LIN {X 0,Y 276.198,Z 756.508,A -85,B 0,C 180,E1 -18193.239,E2 -18193.239} C_VEL
LIN {X 0,Y 277.602,Z 768.151,A -85,B 0,C 180,E1 -18194.665,E2 -18194.665} C_VEL
LIN {X 0,Y 277.773,Z 774.427,A -85,B 0,C 180,E1 -18195.481,E2 -18195.481} C_VEL
LIN {X 0,Y 275.608,Z 785.625,A -85,B 0,C 180,E1 -18196.862,E2 -18196.862} C_VEL
LIN {X 0,Y 273.362,Z 795.783,A -85,B 0,C 180,E1 -18198.433,E2 -18198.433} C_VEL
LIN {X 0,Y 271.104,Z 804.857,A -85,B 0,C 180,E1 -18200.172,E2 -18200.172} C_VEL
LIN {X 0,Y 268.769,Z 813.709,A -85,B 0,C 180,E1 -18202.281,E2 -18202.281} C_VEL
LIN {X 0,Y 266.705,Z 821.184,A -85,B 0,C 180,E1 -18204.521,E2 -18204.521} C_VEL
LIN {X 0,Y 264.933,Z 827.228,A -85,B 0,C 180,E1 -18206.806,E2 -18206.806} C_VEL
LIN {X 0,Y 263.353,Z 832.857,A -85,B 0,C 180,E1 -18209.584,E2 -18209.584} C_VEL
LIN {X 0,Y 262.177,Z 836.929,A -85,B 0,C 180,E1 -18212.42,E2 -18212.42} C_VEL
LIN {X 0,Y 261.591,Z 838.852,A -85,B 0,C 180,E1 -18214.346,E2 -18214.346} C_VEL
LIN {X 0,Y 261.136,Z 840.117,A -85,B 0,C 180,E1 -18216.305,E2 -18216.305} C_VEL
LIN {X 0,Y 260.831,Z 840.792,A -85,B 0,C 180,E1 -18218.613,E2 -18218.613} C_VEL
LIN {X 0,Y 260.686,Z 840.55,A -85,B 0,C 180,E1 -18220.988,E2 -18220.988} C_VEL
LIN {X 0,Y 260.711,Z 839.404,A -85,B 0,C 180,E1 -18223.296,E2 -18223.296} C_VEL
LIN {X 0,Y 260.957,Z 837.388,A -85,B 0,C 180,E1 -18225.557,E2 -18225.557} C_VEL
LIN {X 0,Y 261.385,Z 834.513,A -85,B 0,C 180,E1 -18227.765,E2 -18227.765} C_VEL
LIN {X 0,Y 262.026,Z 829.545,A -85,B 0,C 180,E1 -18230.507,E2 -18230.507} C_VEL
LIN {X 0,Y 262.865,Z 824.396,A -85,B 0,C 180,E1 -18232.688,E2 -18232.688} C_VEL
LIN {X 0,Y 264.105,Z 816.747,A -85,B 0,C 180,E1 -18235.251,E2 -18235.251} C_VEL
LIN {X 0,Y 265.536,Z 808.333,A -85,B 0,C 180,E1 -18237.459,E2 -18237.459} C_VEL
LIN {X 0,Y 267.211,Z 798.256,A -85,B 0,C 180,E1 -18239.584,E2 -18239.584} C_VEL
LIN {X 0,Y 268.75,Z 788.148,A -85,B 0,C 180,E1 -18241.282,E2 -18241.282} C_VEL
LIN {X 0,Y 270.33,Z 776.866,A -85,B 0,C 180,E1 -18242.8,E2 -18242.8} C_VEL
LIN {X 0,Y 271.383,Z 768.818,A -85,B 0,C 180,E1 -18243.675,E2 -18243.675} C_VEL
LIN {X 0,Y 270.234,Z 758.034,A -85,B 0,C 180,E1 -18244.796,E2 -18244.796} C_VEL
LIN {X 0,Y 268.326,Z 744.948,A -85,B 0,C 180,E1 -18245.895,E2 -18245.895} C_VEL
LIN {X 0,Y 265.74,Z 730.76,A -85,B 0,C 180,E1 -18246.793,E2 -18246.793} C_VEL
LIN {X 0,Y 266.686,Z 721.477,A -85,B 0,C 180,E1 -18250.368,E2 -18250.368} C_VEL
LIN {X 0,Y 267.789,Z 710.142,A -85,B 0,C 180,E1 -18254.786,E2 -18254.786} C_VEL
LIN {X 0,Y 268.769,Z 700.139,A -85,B 0,C 180,E1 -18258.691,E2 -18258.691} C_VEL
LIN {X 0,Y 268.925,Z 696.307,A -85,B 0,C 180,E1 -18260.221,E2 -18260.221} C_VEL
LIN {X 0,Y 268.07,Z 689.203,A -85,B 0,C 180,E1 -18263.226,E2 -18263.226} C_VEL
LIN {X 0,Y 266.137,Z 678.968,A -85,B 0,C 180,E1 -18267.731,E2 -18267.731} C_VEL
LIN {X 0,Y 264.857,Z 672.26,A -85,B 0,C 180,E1 -18270.761,E2 -18270.761} C_VEL
LIN {X 0,Y 263.59,Z 667.651,A -85,B 0,C 180,E1 -18272.962,E2 -18272.962} C_VEL
LIN {X 0,Y 263.571,Z 667.653,A -85,B 0,C 180,E1 -18277.662,E2 -18277.662} C_VEL
LIN {X 0,Y 263.376,Z 667.675,A -85,B 0,C 180,E1 -18280.766,E2 -18280.766} C_VEL
LIN {X 0,Y 263.321,Z 667.687,A -85,B 0,C 180,E1 -18283.064,E2 -18283.064} C_VEL
LIN {X 0,Y 267.262,Z 679.189,A -85,B 0,C 180,E1 -18284.467,E2 -18284.467} C_VEL
LIN {X 0,Y 270.498,Z 689.858,A -85,B 0,C 180,E1 -18285.988,E2 -18285.988} C_VEL
LIN {X 0,Y 272.248,Z 696.742,A -85,B 0,C 180,E1 -18287.086,E2 -18287.086} C_VEL
LIN {X 0,Y 271.831,Z 701.91,A -85,B 0,C 180,E1 -18287.861,E2 -18287.861} C_VEL
LIN {X 0,Y 270.282,Z 712.896,A -85,B 0,C 180,E1 -18289.758,E2 -18289.758} C_VEL
LIN {X 0,Y 269.071,Z 720.859,A -85,B 0,C 180,E1 -18291.45,E2 -18291.45} C_VEL
LIN {X 0,Y 267.632,Z 729.101,A -85,B 0,C 180,E1 -18293.566,E2 -18293.566} C_VEL
LIN {X 0,Y 266.612,Z 735.353,A -85,B 0,C 180,E1 -18295.547,E2 -18295.547} C_VEL
LIN {X 0,Y 265.678,Z 740.632,A -85,B 0,C 180,E1 -18297.577,E2 -18297.577} C_VEL
LIN {X 0,Y 264.787,Z 746.106,A -85,B 0,C 180,E1 -18300.286,E2 -18300.286} C_VEL
LIN {X 0,Y 264.073,Z 750.203,A -85,B 0,C 180,E1 -18303.065,E2 -18303.065} C_VEL
LIN {X 0,Y 263.714,Z 752.906,A -85,B 0,C 180,E1 -18305.896,E2 -18305.896} C_VEL
LIN {X 0,Y 263.699,Z 753.93,A -85,B 0,C 180,E1 -18307.806,E2 -18307.806} C_VEL
LIN {X 0,Y 263.903,Z 754.344,A -85,B 0,C 180,E1 -18309.729,E2 -18309.729} C_VEL
LIN {X 0,Y 264.304,Z 754.095,A -85,B 0,C 180,E1 -18311.881,E2 -18311.881} C_VEL
LIN {X 0,Y 264.978,Z 752.884,A -85,B 0,C 180,E1 -18314.265,E2 -18314.265} C_VEL
LIN {X 0,Y 265.878,Z 750.741,A -85,B 0,C 180,E1 -18316.586,E2 -18316.586} C_VEL
LIN {X 0,Y 267.047,Z 747.643,A -85,B 0,C 180,E1 -18318.857,E2 -18318.857} C_VEL
LIN {X 0,Y 268.358,Z 743.632,A -85,B 0,C 180,E1 -18321.058,E2 -18321.058} C_VEL
LIN {X 0,Y 270.359,Z 737.238,A -85,B 0,C 180,E1 -18323.693,E2 -18323.693} C_VEL
LIN {X 0,Y 272.549,Z 729.498,A -85,B 0,C 180,E1 -18326.142,E2 -18326.142} C_VEL
LIN {X 0,Y 274.591,Z 721.267,A -85,B 0,C 180,E1 -18328.186,E2 -18328.186} C_VEL
LIN {X 0,Y 276.931,Z 711.01,A -85,B 0,C 180,E1 -18330.195,E2 -18330.195} C_VEL
LIN {X 0,Y 277.833,Z 706.45,A -85,B 0,C 180,E1 -18330.951,E2 -18330.951} C_VEL
LIN {X 0,Y 275.853,Z 697.824,A -85,B 0,C 180,E1 -18332.704,E2 -18332.704} C_VEL
LIN {X 0,Y 272.997,Z 689.08,A -85,B 0,C 180,E1 -18334.379,E2 -18334.379} C_VEL
LIN {X 0,Y 268.69,Z 678.97,A -85,B 0,C 180,E1 -18336.236,E2 -18336.236} C_VEL
LIN {X 0,Y 264.603,Z 671.132,A -85,B 0,C 180,E1 -18337.657,E2 -18337.657} C_VEL
LIN {X 0,Y 263.299,Z 668.406,A -85,B 0,C 180,E1 -18338.101,E2 -18338.101} C_VEL
LIN {X 0,Y 263.171,Z 667.697,A -85,B 0,C 180,E1 -18338.222,E2 -18338.222} C_VEL
LIN {X 0,Y 263.252,Z 667.697,A -85,B 0,C 180,E1 -18341.315,E2 -18341.315} C_VEL
LIN {X 0,Y 263.353,Z 667.684,A -85,B 0,C 180,E1 -18344.522,E2 -18344.522} C_VEL
LIN {X 0,Y 263.376,Z 667.672,A -85,B 0,C 180,E1 -18349.235,E2 -18349.235} C_VEL
LIN {X 0,Y 263.57,Z 667.642,A -85,B 0,C 180,E1 -18352.394,E2 -18352.394} C_VEL
LIN {X 0,Y 263.754,Z 667.63,A -85,B 0,C 180,E1 -18358.473,E2 -18358.473} C_VEL
LIN {X 0,Y 263.751,Z 667.625,A -85,B 0,C 180,E1 -18359.041,E2 -18359.041} C_VEL
LIN {X 0,Y 263.428,Z 667.663,A -85,B 0,C 180,E1 -18359.893,E2 -18359.893} C_VEL
LIN {X 0,Y 262.001,Z 667.842,A -85,B 0,C 180,E1 -18361.148,E2 -18361.148} C_VEL
LIN {X 0,Y 257.475,Z 668.404,A -85,B 0,C 180,E1 -18364.068,E2 -18364.068} C_VEL
LIN {X 0,Y 256.465,Z 668.526,A -85,B 0,C 180,E1 -18365.379,E2 -18365.379} C_VEL
LIN {X 0,Y 256.426,Z 668.533,A -85,B 0,C 180,E1 -18365.823,E2 -18365.823} C_VEL
LIN {X 0,Y 256.543,Z 668.525,A -85,B 0,C 180,E1 -18367.873,E2 -18367.873} C_VEL
LIN {X 0,Y 256.313,Z 668.558,A -85,B 0,C 180,E1 -18371.066,E2 -18371.066} C_VEL
LIN {X 0,Y 256.303,Z 668.552,A -85,B 0,C 180,E1 -18375.915,E2 -18375.915} C_VEL
LIN {X 0,Y 256.17,Z 668.571,A -85,B 0,C 180,E1 -18380.895,E2 -18380.895} C_VEL
LIN {X 0,Y 256.191,Z 668.57,A -85,B 0,C 180,E1 -18385.138,E2 -18385.138} C_VEL
LIN {X 0,Y 256.113,Z 668.584,A -85,B 0,C 180,E1 -18389.6,E2 -18389.6} C_VEL
LIN {X 0,Y 256.116,Z 668.669,A -85,B 0,C 180,E1 -18390.965,E2 -18390.965} C_VEL
LIN {X 0,Y 257.114,Z 673.07,A -85,B 0,C 180,E1 -18395.031,E2 -18395.031} C_VEL
LIN {X 0,Y 258.119,Z 677.767,A -85,B 0,C 180,E1 -18398.774,E2 -18398.774} C_VEL
LIN {X 0,Y 259.319,Z 683.648,A -85,B 0,C 180,E1 -18402.966,E2 -18402.966} C_VEL
LIN {X 0,Y 260.424,Z 689.622,A -85,B 0,C 180,E1 -18406.773,E2 -18406.773} C_VEL
LIN {X 0,Y 261.295,Z 694.723,A -85,B 0,C 180,E1 -18409.794,E2 -18409.794} C_VEL
LIN {X 0,Y 261.3,Z 697.44,A -85,B 0,C 180,E1 -18411.26,E2 -18411.26} C_VEL
LIN {X 0,Y 259.51,Z 705.627,A -85,B 0,C 180,E1 -18415.338,E2 -18415.338} C_VEL
LIN {X 0,Y 258.309,Z 711.807,A -85,B 0,C 180,E1 -18418.301,E2 -18418.301} C_VEL
LIN {X 0,Y 259.226,Z 715.743,A -85,B 0,C 180,E1 -18418.638,E2 -18418.638} C_VEL
LIN {X 0,Y 262.039,Z 728.793,A -85,B 0,C 180,E1 -18419.914,E2 -18419.914} C_VEL
LIN {X 0,Y 263.696,Z 740.974,A -85,B 0,C 180,E1 -18421.223,E2 -18421.223} C_VEL
LIN {X 0,Y 264.422,Z 753.313,A -85,B 0,C 180,E1 -18422.691,E2 -18422.691} C_VEL
LIN {X 0,Y 264.278,Z 764.335,A -85,B 0,C 180,E1 -18424.184,E2 -18424.184} C_VEL
LIN {X 0,Y 263.493,Z 774.16,A -85,B 0,C 180,E1 -18425.711,E2 -18425.711} C_VEL
LIN {X 0,Y 262.966,Z 778.792,A -85,B 0,C 180,E1 -18426.47,E2 -18426.47} C_VEL
LIN {X 0,Y 262.801,Z 790.833,A -85,B 0,C 180,E1 -18427.806,E2 -18427.806} C_VEL
LIN {X 0,Y 261.376,Z 800.812,A -85,B 0,C 180,E1 -18429.128,E2 -18429.128} C_VEL
LIN {X 0,Y 259.783,Z 811.236,A -85,B 0,C 180,E1 -18430.851,E2 -18430.851} C_VEL
LIN {X 0,Y 258.423,Z 819.807,A -85,B 0,C 180,E1 -18432.593,E2 -18432.593} C_VEL
LIN {X 0,Y 257.094,Z 827.709,A -85,B 0,C 180,E1 -18434.541,E2 -18434.541} C_VEL
LIN {X 0,Y 255.823,Z 835.398,A -85,B 0,C 180,E1 -18436.9,E2 -18436.9} C_VEL
LIN {X 0,Y 254.857,Z 842.458,A -85,B 0,C 180,E1 -18439.673,E2 -18439.673} C_VEL
LIN {X 0,Y 254.389,Z 847.112,A -85,B 0,C 180,E1 -18442.059,E2 -18442.059} C_VEL
LIN {X 0,Y 254.127,Z 850.827,A -85,B 0,C 180,E1 -18444.624,E2 -18444.624} C_VEL
LIN {X 0,Y 254.098,Z 853.059,A -85,B 0,C 180,E1 -18446.828,E2 -18446.828} C_VEL
LIN {X 0,Y 254.127,Z 854.136,A -85,B 0,C 180,E1 -18448.414,E2 -18448.414} C_VEL
LIN {X 0,Y 254.143,Z 854.786,A -85,B 0,C 180,E1 -18449.999,E2 -18449.999} C_VEL
LIN {X 0,Y 254.115,Z 855.035,A -85,B 0,C 180,E1 -18451.584,E2 -18451.584} C_VEL
LIN {X 0,Y 254.053,Z 854.88,A -85,B 0,C 180,E1 -18453.171,E2 -18453.171} C_VEL
LIN {X 0,Y 254.087,Z 854,A -85,B 0,C 180,E1 -18455.278,E2 -18455.278} C_VEL
LIN {X 0,Y 254.388,Z 851.892,A -85,B 0,C 180,E1 -18457.939,E2 -18457.939} C_VEL
LIN {X 0,Y 255.037,Z 848.981,A -85,B 0,C 180,E1 -18460.317,E2 -18460.317} C_VEL
LIN {X 0,Y 255.952,Z 845.067,A -85,B 0,C 180,E1 -18462.688,E2 -18462.688} C_VEL
LIN {X 0,Y 257.305,Z 840.037,A -85,B 0,C 180,E1 -18465.038,E2 -18465.038} C_VEL
LIN {X 0,Y 259.223,Z 833.743,A -85,B 0,C 180,E1 -18467.35,E2 -18467.35} C_VEL
LIN {X 0,Y 261.184,Z 825.971,A -85,B 0,C 180,E1 -18469.645,E2 -18469.645} C_VEL
LIN {X 0,Y 263.83,Z 816.307,A -85,B 0,C 180,E1 -18471.896,E2 -18471.896} C_VEL
LIN {X 0,Y 266.431,Z 806.398,A -85,B 0,C 180,E1 -18473.719,E2 -18473.719} C_VEL
LIN {X 0,Y 268.608,Z 796.768,A -85,B 0,C 180,E1 -18475.161,E2 -18475.161} C_VEL
LIN {X 0,Y 269.759,Z 786.392,A -85,B 0,C 180,E1 -18476.541,E2 -18476.541} C_VEL
LIN {X 0,Y 270.72,Z 774.185,A -85,B 0,C 180,E1 -18477.857,E2 -18477.857} C_VEL
LIN {X 0,Y 270.16,Z 761.918,A -85,B 0,C 180,E1 -18479.06,E2 -18479.06} C_VEL
LIN {X 0,Y 268.281,Z 749.793,A -85,B 0,C 180,E1 -18480.176,E2 -18480.176} C_VEL
LIN {X 0,Y 265.255,Z 737.177,A -85,B 0,C 180,E1 -18481.361,E2 -18481.361} C_VEL
LIN {X 0,Y 265.149,Z 724.817,A -85,B 0,C 180,E1 -18483.998,E2 -18483.998} C_VEL
LIN {X 0,Y 265.153,Z 712.44,A -85,B 0,C 180,E1 -18487.059,E2 -18487.059} C_VEL
LIN {X 0,Y 265.308,Z 702.912,A -85,B 0,C 180,E1 -18489.806,E2 -18489.806} C_VEL
LIN {X 0,Y 263.847,Z 695.598,A -85,B 0,C 180,E1 -18492.904,E2 -18492.904} C_VEL
LIN {X 0,Y 262.817,Z 689.845,A -85,B 0,C 180,E1 -18495.951,E2 -18495.951} C_VEL
LIN {X 0,Y 262.349,Z 685.648,A -85,B 0,C 180,E1 -18498.596,E2 -18498.596} C_VEL
LIN {X 0,Y 262.311,Z 682.419,A -85,B 0,C 180,E1 -18500.984,E2 -18500.984} C_VEL
LIN {X 0,Y 262.124,Z 681.504,A -85,B 0,C 180,E1 -18501.926,E2 -18501.926} C_VEL
LIN {X 0,Y 261.594,Z 680.38,A -85,B 0,C 180,E1 -18503.768,E2 -18503.768} C_VEL
LIN {X 0,Y 260.703,Z 679.193,A -85,B 0,C 180,E1 -18507.373,E2 -18507.373} C_VEL
LIN {X 0,Y 260.545,Z 678.921,A -85,B 0,C 180,E1 -18510.952,E2 -18510.952} C_VEL
LIN {X 0,Y 260.897,Z 679.524,A -85,B 0,C 180,E1 -18514.468,E2 -18514.468} C_VEL
LIN {X 0,Y 261.33,Z 681.273,A -85,B 0,C 180,E1 -18517.882,E2 -18517.882} C_VEL
LIN {X 0,Y 262.144,Z 683.553,A -85,B 0,C 180,E1 -18521.233,E2 -18521.233} C_VEL
LIN {X 0,Y 263.103,Z 686.63,A -85,B 0,C 180,E1 -18524.507,E2 -18524.507} C_VEL
LIN {X 0,Y 264.179,Z 690.307,A -85,B 0,C 180,E1 -18527.712,E2 -18527.712} C_VEL
LIN {X 0,Y 265.301,Z 694.517,A -85,B 0,C 180,E1 -18530.854,E2 -18530.854} C_VEL
LIN {X 0,Y 265.917,Z 698.003,A -85,B 0,C 180,E1 -18533.169,E2 -18533.169} C_VEL
LIN {X 0,Y 267.075,Z 704.475,A -85,B 0,C 180,E1 -18536.983,E2 -18536.983} C_VEL
LIN {X 0,Y 267.344,Z 708.812,A -85,B 0,C 180,E1 -18539.247,E2 -18539.247} C_VEL
LIN {X 0,Y 266.872,Z 713.663,A -85,B 0,C 180,E1 -18541.509,E2 -18541.509} C_VEL
LIN {X 0,Y 265.153,Z 722.566,A -85,B 0,C 180,E1 -18545.323,E2 -18545.323} C_VEL
LIN {X 0,Y 263.557,Z 732.414,A -85,B 0,C 180,E1 -18549.433,E2 -18549.433} C_VEL
LIN {X 0,Y 267.559,Z 745.4,A -85,B 0,C 180,E1 -18550.926,E2 -18550.926} C_VEL
LIN {X 0,Y 269.966,Z 756.451,A -85,B 0,C 180,E1 -18552.259,E2 -18552.259} C_VEL
LIN {X 0,Y 271.458,Z 768.872,A -85,B 0,C 180,E1 -18553.856,E2 -18553.856} C_VEL
LIN {X 0,Y 271.578,Z 776.267,A -85,B 0,C 180,E1 -18554.854,E2 -18554.854} C_VEL
LIN {X 0,Y 269.44,Z 786.352,A -85,B 0,C 180,E1 -18556.138,E2 -18556.138} C_VEL
LIN {X 0,Y 266.947,Z 796.894,A -85,B 0,C 180,E1 -18557.838,E2 -18557.838} C_VEL
LIN {X 0,Y 264.334,Z 806.704,A -85,B 0,C 180,E1 -18559.815,E2 -18559.815} C_VEL
LIN {X 0,Y 261.823,Z 815.559,A -85,B 0,C 180,E1 -18562.073,E2 -18562.073} C_VEL
LIN {X 0,Y 259.708,Z 822.713,A -85,B 0,C 180,E1 -18564.373,E2 -18564.373} C_VEL
LIN {X 0,Y 257.793,Z 828.767,A -85,B 0,C 180,E1 -18566.829,E2 -18566.829} C_VEL
LIN {X 0,Y 256.254,Z 833.863,A -85,B 0,C 180,E1 -18569.582,E2 -18569.582} C_VEL
LIN {X 0,Y 255.073,Z 837.663,A -85,B 0,C 180,E1 -18572.499,E2 -18572.499} C_VEL
LIN {X 0,Y 254.223,Z 840.08,A -85,B 0,C 180,E1 -18575.489,E2 -18575.489} C_VEL
LIN {X 0,Y 253.845,Z 840.865,A -85,B 0,C 180,E1 -18577.524,E2 -18577.524} C_VEL
LIN {X 0,Y 253.65,Z 841,A -85,B 0,C 180,E1 -18579.588,E2 -18579.588} C_VEL
LIN {X 0,Y 253.574,Z 840.459,A -85,B 0,C 180,E1 -18581.696,E2 -18581.696} C_VEL
LIN {X 0,Y 253.747,Z 838.174,A -85,B 0,C 180,E1 -18584.931,E2 -18584.931} C_VEL
LIN {X 0,Y 254.159,Z 835.56,A -85,B 0,C 180,E1 -18587.173,E2 -18587.173} C_VEL
LIN {X 0,Y 254.667,Z 831.764,A -85,B 0,C 180,E1 -18589.561,E2 -18589.561} C_VEL
LIN {X 0,Y 255.582,Z 826.036,A -85,B 0,C 180,E1 -18592.279,E2 -18592.279} C_VEL
LIN {X 0,Y 256.784,Z 818.721,A -85,B 0,C 180,E1 -18594.919,E2 -18594.919} C_VEL
LIN {X 0,Y 258.065,Z 811.51,A -85,B 0,C 180,E1 -18596.999,E2 -18596.999} C_VEL
LIN {X 0,Y 259.527,Z 802.88,A -85,B 0,C 180,E1 -18599.036,E2 -18599.036} C_VEL
LIN {X 0,Y 261.293,Z 792.219,A -85,B 0,C 180,E1 -18601.045,E2 -18601.045} C_VEL
LIN {X 0,Y 263.059,Z 780.544,A -85,B 0,C 180,E1 -18602.791,E2 -18602.791} C_VEL
LIN {X 0,Y 264.555,Z 769.194,A -85,B 0,C 180,E1 -18604.11,E2 -18604.11} C_VEL
LIN {X 0,Y 263.244,Z 757.596,A -85,B 0,C 180,E1 -18605.345,E2 -18605.345} C_VEL
LIN {X 0,Y 261.369,Z 744.354,A -85,B 0,C 180,E1 -18606.461,E2 -18606.461} C_VEL
LIN {X 0,Y 258.895,Z 730.821,A -85,B 0,C 180,E1 -18607.363,E2 -18607.363} C_VEL
LIN {X 0,Y 259.913,Z 721.187,A -85,B 0,C 180,E1 -18611.154,E2 -18611.154} C_VEL
LIN {X 0,Y 261.073,Z 709.657,A -85,B 0,C 180,E1 -18615.721,E2 -18615.721} C_VEL
LIN {X 0,Y 261.955,Z 700.966,A -85,B 0,C 180,E1 -18619.176,E2 -18619.176} C_VEL
LIN {X 0,Y 262.004,Z 697.167,A -85,B 0,C 180,E1 -18620.739,E2 -18620.739} C_VEL
LIN {X 0,Y 261.072,Z 690.061,A -85,B 0,C 180,E1 -18623.819,E2 -18623.819} C_VEL
LIN {X 0,Y 258.917,Z 678.058,A -85,B 0,C 180,E1 -18629.223,E2 -18629.223} C_VEL
LIN {X 0,Y 257.328,Z 671.447,A -85,B 0,C 180,E1 -18632.349,E2 -18632.349} C_VEL
LIN {X 0,Y 256.431,Z 668.538,A -85,B 0,C 180,E1 -18633.831,E2 -18633.831} C_VEL
LIN {X 0,Y 256.539,Z 668.531,A -85,B 0,C 180,E1 -18637.874,E2 -18637.874} C_VEL
LIN {X 0,Y 256.298,Z 668.565,A -85,B 0,C 180,E1 -18642.472,E2 -18642.472} C_VEL
LIN {X 0,Y 260.16,Z 679.738,A -85,B 0,C 180,E1 -18643.873,E2 -18643.873} C_VEL
LIN {X 0,Y 263.807,Z 691.758,A -85,B 0,C 180,E1 -18645.649,E2 -18645.649} C_VEL
LIN {X 0,Y 265.526,Z 699.429,A -85,B 0,C 180,E1 -18646.928,E2 -18646.928} C_VEL
LIN {X 0,Y 264.098,Z 709.824,A -85,B 0,C 180,E1 -18648.623,E2 -18648.623} C_VEL
LIN {X 0,Y 262.641,Z 719.226,A -85,B 0,C 180,E1 -18650.518,E2 -18650.518} C_VEL
LIN {X 0,Y 261.043,Z 728.359,A -85,B 0,C 180,E1 -18652.809,E2 -18652.809} C_VEL
LIN {X 0,Y 259.706,Z 736.071,A -85,B 0,C 180,E1 -18655.228,E2 -18655.228} C_VEL
LIN {X 0,Y 258.652,Z 741.864,A -85,B 0,C 180,E1 -18657.512,E2 -18657.512} C_VEL
LIN {X 0,Y 257.76,Z 747.287,A -85,B 0,C 180,E1 -18660.293,E2 -18660.293} C_VEL
LIN {X 0,Y 257.03,Z 751.359,A -85,B 0,C 180,E1 -18663.153,E2 -18663.153} C_VEL
LIN {X 0,Y 256.741,Z 753.268,A -85,B 0,C 180,E1 -18665.09,E2 -18665.09} C_VEL
LIN {X 0,Y 256.661,Z 754.769,A -85,B 0,C 180,E1 -18667.431,E2 -18667.431} C_VEL
LIN {X 0,Y 256.915,Z 755.394,A -85,B 0,C 180,E1 -18670.009,E2 -18670.009} C_VEL
LIN {X 0,Y 257.575,Z 754.802,A -85,B 0,C 180,E1 -18673.011,E2 -18673.011} C_VEL
LIN {X 0,Y 258.228,Z 753.567,A -85,B 0,C 180,E1 -18675.043,E2 -18675.043} C_VEL
LIN {X 0,Y 259.684,Z 750.335,A -85,B 0,C 180,E1 -18678.147,E2 -18678.147} C_VEL
LIN {X 0,Y 260.915,Z 746.943,A -85,B 0,C 180,E1 -18680.347,E2 -18680.347} C_VEL
LIN {X 0,Y 262.401,Z 742.612,A -85,B 0,C 180,E1 -18682.504,E2 -18682.504} C_VEL
LIN {X 0,Y 264.441,Z 736.134,A -85,B 0,C 180,E1 -18685.011,E2 -18685.011} C_VEL
LIN {X 0,Y 266.839,Z 727.964,A -85,B 0,C 180,E1 -18687.439,E2 -18687.439} C_VEL
LIN {X 0,Y 268.937,Z 719.787,A -85,B 0,C 180,E1 -18689.386,E2 -18689.386} C_VEL
LIN {X 0,Y 271.182,Z 709.87,A -85,B 0,C 180,E1 -18691.267,E2 -18691.267} C_VEL
LIN {X 0,Y 271.362,Z 707.49,A -85,B 0,C 180,E1 -18691.711,E2 -18691.711} C_VEL
LIN {X 0,Y 269.1,Z 698.473,A -85,B 0,C 180,E1 -18693.642,E2 -18693.642} C_VEL
LIN {X 0,Y 266.097,Z 689.627,A -85,B 0,C 180,E1 -18695.419,E2 -18695.419} C_VEL
LIN {X 0,Y 262.296,Z 680.843,A -85,B 0,C 180,E1 -18697.138,E2 -18697.138} C_VEL
LIN {X 0,Y 257.795,Z 672.308,A -85,B 0,C 180,E1 -18698.79,E2 -18698.79} C_VEL
LIN {X 0,Y 256.41,Z 669.572,A -85,B 0,C 180,E1 -18699.283,E2 -18699.283} C_VEL
LIN {X 0,Y 256.211,Z 668.576,A -85,B 0,C 180,E1 -18699.424,E2 -18699.424} C_VEL
LIN {X 0,Y 256.303,Z 668.564,A -85,B 0,C 180,E1 -18704.085,E2 -18704.085} C_VEL
LIN {X 0,Y 256.312,Z 668.551,A -85,B 0,C 180,E1 -18708.934,E2 -18708.934} C_VEL
LIN {X 0,Y 256.542,Z 668.518,A -85,B 0,C 180,E1 -18712.127,E2 -18712.127} C_VEL
LIN {X 0,Y 256.717,Z 668.506,A -85,B 0,C 180,E1 -18718.431,E2 -18718.431} C_VEL
LIN {X 0,Y 256.717,Z 668.495,A -85,B 0,C 180,E1 -18721.569,E2 -18721.569} C_VEL
LIN {X 0,Y 256.426,Z 668.533,A -85,B 0,C 180,E1 -18725.823,E2 -18725.823} C_VEL
LIN {X 0,Y 255.843,Z 668.616,A -85,B 0,C 180,E1 -18727.134,E2 -18727.134} C_VEL
LIN {X 0,Y 254.241,Z 668.816,A -85,B 0,C 180,E1 -18728.419,E2 -18728.419} C_VEL
LIN {X 0,Y 250.37,Z 669.299,A -85,B 0,C 180,E1 -18731.003,E2 -18731.003} C_VEL
LIN {X 0,Y 249.293,Z 669.424,A -85,B 0,C 180,E1 -18732.354,E2 -18732.354} C_VEL
LIN {X 0,Y 249.217,Z 669.431,A -85,B 0,C 180,E1 -18732.813,E2 -18732.813} C_VEL
LIN {X 0,Y 249.221,Z 669.432,A -85,B 0,C 180,E1 -18736.503,E2 -18736.503} C_VEL
LIN {X 0,Y 249.09,Z 669.458,A -85,B 0,C 180,E1 -18741.518,E2 -18741.518} C_VEL
LIN {X 0,Y 249.133,Z 669.447,A -85,B 0,C 180,E1 -18745.482,E2 -18745.482} C_VEL
LIN {X 0,Y 249.079,Z 669.481,A -85,B 0,C 180,E1 -18749.465,E2 -18749.465} C_VEL
LIN {X 0,Y 250.109,Z 674.299,A -85,B 0,C 180,E1 -18754.194,E2 -18754.194} C_VEL
LIN {X 0,Y 251.158,Z 678.806,A -85,B 0,C 180,E1 -18757.997,E2 -18757.997} C_VEL
LIN {X 0,Y 252.229,Z 684.127,A -85,B 0,C 180,E1 -18761.969,E2 -18761.969} C_VEL
LIN {X 0,Y 253.387,Z 690.369,A -85,B 0,C 180,E1 -18766.149,E2 -18766.149} C_VEL
LIN {X 0,Y 254.311,Z 695.85,A -85,B 0,C 180,E1 -18769.5,E2 -18769.5} C_VEL
LIN {X 0,Y 254.424,Z 697.863,A -85,B 0,C 180,E1 -18770.665,E2 -18770.665} C_VEL
LIN {X 0,Y 253.189,Z 703.541,A -85,B 0,C 180,E1 -18773.609,E2 -18773.609} C_VEL
LIN {X 0,Y 251.724,Z 710.396,A -85,B 0,C 180,E1 -18777.065,E2 -18777.065} C_VEL
LIN {X 0,Y 252.588,Z 714.261,A -85,B 0,C 180,E1 -18777.418,E2 -18777.418} C_VEL
LIN {X 0,Y 255.785,Z 728.79,A -85,B 0,C 180,E1 -18778.963,E2 -18778.963} C_VEL
LIN {X 0,Y 257.465,Z 741.904,A -85,B 0,C 180,E1 -18780.458,E2 -18780.458} C_VEL
LIN {X 0,Y 258.018,Z 753.769,A -85,B 0,C 180,E1 -18781.962,E2 -18781.962} C_VEL
LIN {X 0,Y 257.707,Z 765.764,A -85,B 0,C 180,E1 -18783.694,E2 -18783.694} C_VEL
LIN {X 0,Y 256.678,Z 776.105,A -85,B 0,C 180,E1 -18785.42,E2 -18785.42} C_VEL
LIN {X 0,Y 256.143,Z 779.967,A -85,B 0,C 180,E1 -18786.127,E2 -18786.127} C_VEL
LIN {X 0,Y 255.832,Z 792.407,A -85,B 0,C 180,E1 -18787.594,E2 -18787.594} C_VEL
LIN {X 0,Y 254.063,Z 803.304,A -85,B 0,C 180,E1 -18789.135,E2 -18789.135} C_VEL
LIN {X 0,Y 252.475,Z 813.438,A -85,B 0,C 180,E1 -18790.953,E2 -18790.953} C_VEL
LIN {X 0,Y 251.08,Z 822.243,A -85,B 0,C 180,E1 -18792.907,E2 -18792.907} C_VEL
LIN {X 0,Y 249.5,Z 831.021,A -85,B 0,C 180,E1 -18795.314,E2 -18795.314} C_VEL
LIN {X 0,Y 248.342,Z 838.008,A -85,B 0,C 180,E1 -18797.745,E2 -18797.745} C_VEL
LIN {X 0,Y 247.635,Z 843.577,A -85,B 0,C 180,E1 -18800.195,E2 -18800.195} C_VEL
LIN {X 0,Y 247.204,Z 847.908,A -85,B 0,C 180,E1 -18802.649,E2 -18802.649} C_VEL
LIN {X 0,Y 247.012,Z 851.123,A -85,B 0,C 180,E1 -18805.103,E2 -18805.103} C_VEL
LIN {X 0,Y 247.013,Z 852.703,A -85,B 0,C 180,E1 -18806.737,E2 -18806.737} C_VEL
LIN {X 0,Y 247.054,Z 853.848,A -85,B 0,C 180,E1 -18808.369,E2 -18808.369} C_VEL
LIN {X 0,Y 247.069,Z 854.533,A -85,B 0,C 180,E1 -18809.999,E2 -18809.999} C_VEL
LIN {X 0,Y 247.041,Z 854.815,A -85,B 0,C 180,E1 -18811.629,E2 -18811.629} C_VEL
LIN {X 0,Y 246.952,Z 854.699,A -85,B 0,C 180,E1 -18813.262,E2 -18813.262} C_VEL
LIN {X 0,Y 246.991,Z 854.01,A -85,B 0,C 180,E1 -18815.181,E2 -18815.181} C_VEL
LIN {X 0,Y 247.35,Z 851.85,A -85,B 0,C 180,E1 -18818.166,E2 -18818.166} C_VEL
LIN {X 0,Y 248.017,Z 849.025,A -85,B 0,C 180,E1 -18820.613,E2 -18820.613} C_VEL
LIN {X 0,Y 248.993,Z 845.193,A -85,B 0,C 180,E1 -18823.049,E2 -18823.049} C_VEL
LIN {X 0,Y 250.458,Z 840.248,A -85,B 0,C 180,E1 -18825.46,E2 -18825.46} C_VEL
LIN {X 0,Y 252.451,Z 834.059,A -85,B 0,C 180,E1 -18827.831,E2 -18827.831} C_VEL
LIN {X 0,Y 254.471,Z 826.743,A -85,B 0,C 180,E1 -18830.112,E2 -18830.112} C_VEL
LIN {X 0,Y 257.302,Z 817.019,A -85,B 0,C 180,E1 -18832.481,E2 -18832.481} C_VEL
LIN {X 0,Y 260.008,Z 807.363,A -85,B 0,C 180,E1 -18834.342,E2 -18834.342} C_VEL
LIN {X 0,Y 262.479,Z 796.669,A -85,B 0,C 180,E1 -18836.004,E2 -18836.004} C_VEL
LIN {X 0,Y 263.988,Z 784.487,A -85,B 0,C 180,E1 -18837.635,E2 -18837.635} C_VEL
LIN {X 0,Y 264.832,Z 772.742,A -85,B 0,C 180,E1 -18838.925,E2 -18838.925} C_VEL
LIN {X 0,Y 264.107,Z 760.842,A -85,B 0,C 180,E1 -18840.154,E2 -18840.154} C_VEL
LIN {X 0,Y 262.061,Z 748.446,A -85,B 0,C 180,E1 -18841.351,E2 -18841.351} C_VEL
LIN {X 0,Y 259.277,Z 737.25,A -85,B 0,C 180,E1 -18842.49,E2 -18842.49} C_VEL
LIN {X 0,Y 259.299,Z 726.629,A -85,B 0,C 180,E1 -18844.888,E2 -18844.888} C_VEL
LIN {X 0,Y 259.568,Z 714.608,A -85,B 0,C 180,E1 -18847.991,E2 -18847.991} C_VEL
LIN {X 0,Y 259.855,Z 708.265,A -85,B 0,C 180,E1 -18849.843,E2 -18849.843} C_VEL
LIN {X 0,Y 259.704,Z 705.742,A -85,B 0,C 180,E1 -18850.736,E2 -18850.736} C_VEL
LIN {X 0,Y 258.745,Z 700.938,A -85,B 0,C 180,E1 -18852.83,E2 -18852.83} C_VEL
LIN {X 0,Y 257.873,Z 696.4,A -85,B 0,C 180,E1 -18855.119,E2 -18855.119} C_VEL
LIN {X 0,Y 257.227,Z 690.902,A -85,B 0,C 180,E1 -18858.506,E2 -18858.506} C_VEL
LIN {X 0,Y 257.167,Z 687.403,A -85,B 0,C 180,E1 -18861.056,E2 -18861.056} C_VEL
LIN {X 0,Y 256.671,Z 685.803,A -85,B 0,C 180,E1 -18862.958,E2 -18862.958} C_VEL
LIN {X 0,Y 255.919,Z 684.589,A -85,B 0,C 180,E1 -18865.47,E2 -18865.47} C_VEL
LIN {X 0,Y 255.233,Z 683.652,A -85,B 0,C 180,E1 -18870.288,E2 -18870.288} C_VEL
LIN {X 0,Y 255.429,Z 684.042,A -85,B 0,C 180,E1 -18873.881,E2 -18873.881} C_VEL
LIN {X 0,Y 255.75,Z 685.505,A -85,B 0,C 180,E1 -18877.373,E2 -18877.373} C_VEL
LIN {X 0,Y 256.433,Z 687.582,A -85,B 0,C 180,E1 -18880.799,E2 -18880.799} C_VEL
LIN {X 0,Y 257.247,Z 690.441,A -85,B 0,C 180,E1 -18884.145,E2 -18884.145} C_VEL
LIN {X 0,Y 258.474,Z 694.968,A -85,B 0,C 180,E1 -18888.189,E2 -18888.189} C_VEL
LIN {X 0,Y 259.545,Z 699.239,A -85,B 0,C 180,E1 -18891.435,E2 -18891.435} C_VEL
LIN {X 0,Y 260.683,Z 706.296,A -85,B 0,C 180,E1 -18895.944,E2 -18895.944} C_VEL
LIN {X 0,Y 261.008,Z 710.798,A -85,B 0,C 180,E1 -18898.457,E2 -18898.457} C_VEL
LIN {X 0,Y 260.618,Z 715.705,A -85,B 0,C 180,E1 -18900.86,E2 -18900.86} C_VEL
LIN {X 0,Y 258.829,Z 724.346,A -85,B 0,C 180,E1 -18904.672,E2 -18904.672} C_VEL
LIN {X 0,Y 257.325,Z 732.496,A -85,B 0,C 180,E1 -18908.194,E2 -18908.194} C_VEL
LIN {X 0,Y 261.588,Z 746.147,A -85,B 0,C 180,E1 -18909.901,E2 -18909.901} C_VEL
LIN {X 0,Y 264.179,Z 758.681,A -85,B 0,C 180,E1 -18911.504,E2 -18911.504} C_VEL
LIN {X 0,Y 265.394,Z 769.706,A -85,B 0,C 180,E1 -18913.008,E2 -18913.008} C_VEL
LIN {X 0,Y 265.569,Z 776.41,A -85,B 0,C 180,E1 -18913.974,E2 -18913.974} C_VEL
LIN {X 0,Y 263.143,Z 787.778,A -85,B 0,C 180,E1 -18915.49,E2 -18915.49} C_VEL
LIN {X 0,Y 260.487,Z 798.329,A -85,B 0,C 180,E1 -18917.264,E2 -18917.264} C_VEL
LIN {X 0,Y 258.021,Z 807.039,A -85,B 0,C 180,E1 -18919.078,E2 -18919.078} C_VEL
LIN {X 0,Y 255.373,Z 815.846,A -85,B 0,C 180,E1 -18921.385,E2 -18921.385} C_VEL
LIN {X 0,Y 252.805,Z 823.931,A -85,B 0,C 180,E1 -18924.096,E2 -18924.096} C_VEL
LIN {X 0,Y 250.805,Z 829.785,A -85,B 0,C 180,E1 -18926.638,E2 -18926.638} C_VEL
LIN {X 0,Y 249.384,Z 834.153,A -85,B 0,C 180,E1 -18929.12,E2 -18929.12} C_VEL
LIN {X 0,Y 248.216,Z 837.656,A -85,B 0,C 180,E1 -18931.854,E2 -18931.854} C_VEL
LIN {X 0,Y 247.326,Z 839.979,A -85,B 0,C 180,E1 -18934.633,E2 -18934.633} C_VEL
LIN {X 0,Y 246.801,Z 841.045,A -85,B 0,C 180,E1 -18937.125,E2 -18937.125} C_VEL
LIN {X 0,Y 246.557,Z 841.169,A -85,B 0,C 180,E1 -18939.682,E2 -18939.682} C_VEL
LIN {X 0,Y 246.475,Z 840.354,A -85,B 0,C 180,E1 -18942.154,E2 -18942.154} C_VEL
LIN {X 0,Y 246.721,Z 837.865,A -85,B 0,C 180,E1 -18945.409,E2 -18945.409} C_VEL
LIN {X 0,Y 247.33,Z 833.915,A -85,B 0,C 180,E1 -18948.458,E2 -18948.458} C_VEL
LIN {X 0,Y 247.886,Z 829.883,A -85,B 0,C 180,E1 -18950.735,E2 -18950.735} C_VEL
LIN {X 0,Y 248.794,Z 824.771,A -85,B 0,C 180,E1 -18953.016,E2 -18953.016} C_VEL
LIN {X 0,Y 249.845,Z 818.478,A -85,B 0,C 180,E1 -18955.281,E2 -18955.281} C_VEL
LIN {X 0,Y 251.286,Z 810.697,A -85,B 0,C 180,E1 -18957.545,E2 -18957.545} C_VEL
LIN {X 0,Y 252.961,Z 801.056,A -85,B 0,C 180,E1 -18959.787,E2 -18959.787} C_VEL
LIN {X 0,Y 254.772,Z 790.341,A -85,B 0,C 180,E1 -18961.779,E2 -18961.779} C_VEL
LIN {X 0,Y 256.372,Z 779.859,A -85,B 0,C 180,E1 -18963.329,E2 -18963.329} C_VEL
LIN {X 0,Y 257.69,Z 769.496,A -85,B 0,C 180,E1 -18964.561,E2 -18964.561} C_VEL
LIN {X 0,Y 256.246,Z 756.95,A -85,B 0,C 180,E1 -18965.936,E2 -18965.936} C_VEL
LIN {X 0,Y 254.381,Z 743.77,A -85,B 0,C 180,E1 -18967.059,E2 -18967.059} C_VEL
LIN {X 0,Y 252.026,Z 730.951,A -85,B 0,C 180,E1 -18967.94,E2 -18967.94} C_VEL
LIN {X 0,Y 253.033,Z 721.932,A -85,B 0,C 180,E1 -18971.557,E2 -18971.557} C_VEL
LIN {X 0,Y 254.154,Z 711.382,A -85,B 0,C 180,E1 -18975.806,E2 -18975.806} C_VEL
LIN {X 0,Y 255.147,Z 701.799,A -85,B 0,C 180,E1 -18979.687,E2 -18979.687} C_VEL
LIN {X 0,Y 254.879,Z 696.217,A -85,B 0,C 180,E1 -18982.076,E2 -18982.076} C_VEL
LIN {X 0,Y 253.728,Z 689.188,A -85,B 0,C 180,E1 -18985.234,E2 -18985.234} C_VEL
LIN {X 0,Y 251.939,Z 678.854,A -85,B 0,C 180,E1 -18990.001,E2 -18990.001} C_VEL
LIN {X 0,Y 250.157,Z 672.291,A -85,B 0,C 180,E1 -18993.222,E2 -18993.222} C_VEL
LIN {X 0,Y 249.318,Z 669.428,A -85,B 0,C 180,E1 -18994.751,E2 -18994.751} C_VEL
LIN {X 0,Y 249.479,Z 669.411,A -85,B 0,C 180,E1 -18998.098,E2 -18998.098} C_VEL
LIN {X 0,Y 249.267,Z 669.436,A -85,B 0,C 180,E1 -19001.847,E2 -19001.847} C_VEL
LIN {X 0,Y 253.454,Z 681.482,A -85,B 0,C 180,E1 -19003.428,E2 -19003.428} C_VEL
LIN {X 0,Y 256.944,Z 693.121,A -85,B 0,C 180,E1 -19005.204,E2 -19005.204} C_VEL
LIN {X 0,Y 258.725,Z 701.004,A -85,B 0,C 180,E1 -19006.573,E2 -19006.573} C_VEL
LIN {X 0,Y 257.307,Z 710.835,A -85,B 0,C 180,E1 -19008.225,E2 -19008.225} C_VEL
LIN {X 0,Y 255.858,Z 719.866,A -85,B 0,C 180,E1 -19010.082,E2 -19010.082} C_VEL
LIN {X 0,Y 254.279,Z 728.733,A -85,B 0,C 180,E1 -19012.337,E2 -19012.337} C_VEL
LIN {X 0,Y 252.936,Z 736.029,A -85,B 0,C 180,E1 -19014.633,E2 -19014.633} C_VEL
LIN {X 0,Y 251.899,Z 741.559,A -85,B 0,C 180,E1 -19016.773,E2 -19016.773} C_VEL
LIN {X 0,Y 251.077,Z 746.321,A -85,B 0,C 180,E1 -19019.06,E2 -19019.06} C_VEL
LIN {X 0,Y 250.427,Z 749.971,A -85,B 0,C 180,E1 -19021.278,E2 -19021.278} C_VEL
LIN {X 0,Y 249.815,Z 753.517,A -85,B 0,C 180,E1 -19024.24,E2 -19024.24} C_VEL
LIN {X 0,Y 249.644,Z 755.107,A -85,B 0,C 180,E1 -19026.242,E2 -19026.242} C_VEL
LIN {X 0,Y 249.696,Z 756.1,A -85,B 0,C 180,E1 -19028.26,E2 -19028.26} C_VEL
LIN {X 0,Y 250.013,Z 756.45,A -85,B 0,C 180,E1 -19030.626,E2 -19030.626} C_VEL
LIN {X 0,Y 250.611,Z 755.898,A -85,B 0,C 180,E1 -19033.187,E2 -19033.187} C_VEL
LIN {X 0,Y 251.468,Z 754.397,A -85,B 0,C 180,E1 -19035.678,E2 -19035.678} C_VEL
LIN {X 0,Y 252.908,Z 751.336,A -85,B 0,C 180,E1 -19038.617,E2 -19038.617} C_VEL
LIN {X 0,Y 254.139,Z 748.141,A -85,B 0,C 180,E1 -19040.744,E2 -19040.744} C_VEL
LIN {X 0,Y 256.071,Z 742.866,A -85,B 0,C 180,E1 -19043.397,E2 -19043.397} C_VEL
LIN {X 0,Y 258.393,Z 735.868,A -85,B 0,C 180,E1 -19046.054,E2 -19046.054} C_VEL
LIN {X 0,Y 260.671,Z 728.366,A -85,B 0,C 180,E1 -19048.283,E2 -19048.283} C_VEL
LIN {X 0,Y 263.045,Z 719.468,A -85,B 0,C 180,E1 -19050.379,E2 -19050.379} C_VEL
LIN {X 0,Y 265.102,Z 710.218,A -85,B 0,C 180,E1 -19052.144,E2 -19052.144} C_VEL
LIN {X 0,Y 262.914,Z 700.868,A -85,B 0,C 180,E1 -19054.254,E2 -19054.254} C_VEL
LIN {X 0,Y 260.055,Z 692.369,A -85,B 0,C 180,E1 -19056.086,E2 -19056.086} C_VEL
LIN {X 0,Y 255.737,Z 682.389,A -85,B 0,C 180,E1 -19058.171,E2 -19058.171} C_VEL
LIN {X 0,Y 250.988,Z 673.386,A -85,B 0,C 180,E1 -19060.046,E2 -19060.046} C_VEL
LIN {X 0,Y 249.394,Z 670.633,A -85,B 0,C 180,E1 -19060.61,E2 -19060.61} C_VEL
LIN {X 0,Y 249.142,Z 669.452,A -85,B 0,C 180,E1 -19060.804,E2 -19060.804} C_VEL
LIN {X 0,Y 249.245,Z 669.439,A -85,B 0,C 180,E1 -19063.622,E2 -19063.622} C_VEL
LIN {X 0,Y 249.255,Z 669.43,A -85,B 0,C 180,E1 -19068.617,E2 -19068.617} C_VEL
LIN {X 0,Y 249.484,Z 669.398,A -85,B 0,C 180,E1 -19071.903,E2 -19071.903} C_VEL
LIN {X 0,Y 249.439,Z 669.4,A -85,B 0,C 180,E1 -19076.77,E2 -19076.77} C_VEL
LIN {X 0,Y 249.731,Z 669.368,A -85,B 0,C 180,E1 -19080,E2 -19080} C_VEL
LIN {X 0,Y 249.44,Z 669.413,A -85,B 0,C 180,E1 -19083.231,E2 -19083.231} C_VEL
LIN {X 0,Y 249.484,Z 669.401,A -85,B 0,C 180,E1 -19088.097,E2 -19088.097} C_VEL
LIN {X 0,Y 249.256,Z 669.437,A -85,B 0,C 180,E1 -19091.384,E2 -19091.384} C_VEL
LIN {X 0,Y 249.217,Z 669.431,A -85,B 0,C 180,E1 -19092.813,E2 -19092.813} C_VEL
LIN {X 0,Y 248.562,Z 669.522,A -85,B 0,C 180,E1 -19094.161,E2 -19094.161} C_VEL
LIN {X 0,Y 245.645,Z 669.877,A -85,B 0,C 180,E1 -19096.357,E2 -19096.357} C_VEL
LIN {X 0,Y 243.159,Z 670.196,A -85,B 0,C 180,E1 -19098.146,E2 -19098.146} C_VEL
LIN {X 0,Y 242.106,Z 670.32,A -85,B 0,C 180,E1 -19099.536,E2 -19099.536} C_VEL
LIN {X 0,Y 242.029,Z 670.328,A -85,B 0,C 180,E1 -19100.008,E2 -19100.008} C_VEL
LIN {X 0,Y 242.06,Z 670.33,A -85,B 0,C 180,E1 -19103.984,E2 -19103.984} C_VEL
LIN {X 0,Y 242.026,Z 670.402,A -85,B 0,C 180,E1 -19107.921,E2 -19107.921} C_VEL
LIN {X 0,Y 242.724,Z 673.621,A -85,B 0,C 180,E1 -19111.412,E2 -19111.412} C_VEL
LIN {X 0,Y 243.924,Z 678.757,A -85,B 0,C 180,E1 -19116.22,E2 -19116.22} C_VEL
LIN {X 0,Y 244.927,Z 683.697,A -85,B 0,C 180,E1 -19120.213,E2 -19120.213} C_VEL
LIN {X 0,Y 246.054,Z 689.549,A -85,B 0,C 180,E1 -19124.432,E2 -19124.432} C_VEL
LIN {X 0,Y 247.138,Z 695.72,A -85,B 0,C 180,E1 -19128.447,E2 -19128.447} C_VEL
LIN {X 0,Y 247.427,Z 699.5,A -85,B 0,C 180,E1 -19130.699,E2 -19130.699} C_VEL
LIN {X 0,Y 245.893,Z 705.952,A -85,B 0,C 180,E1 -19134.131,E2 -19134.131} C_VEL
LIN {X 0,Y 245.22,Z 709.031,A -85,B 0,C 180,E1 -19135.736,E2 -19135.736} C_VEL
LIN {X 0,Y 246.06,Z 712.868,A -85,B 0,C 180,E1 -19136.119,E2 -19136.119} C_VEL
LIN {X 0,Y 249.145,Z 726.123,A -85,B 0,C 180,E1 -19137.627,E2 -19137.627} C_VEL
LIN {X 0,Y 250.949,Z 739.35,A -85,B 0,C 180,E1 -19139.22,E2 -19139.22} C_VEL
LIN {X 0,Y 251.61,Z 751.222,A -85,B 0,C 180,E1 -19140.769,E2 -19140.769} C_VEL
LIN {X 0,Y 251.429,Z 763.153,A -85,B 0,C 180,E1 -19142.534,E2 -19142.534} C_VEL
LIN {X 0,Y 250.327,Z 774.574,A -85,B 0,C 180,E1 -19144.482,E2 -19144.482} C_VEL
LIN {X 0,Y 249.312,Z 781.508,A -85,B 0,C 180,E1 -19145.818,E2 -19145.818} C_VEL
LIN {X 0,Y 248.971,Z 792.414,A -85,B 0,C 180,E1 -19147.161,E2 -19147.161} C_VEL
LIN {X 0,Y 247.187,Z 803.277,A -85,B 0,C 180,E1 -19148.745,E2 -19148.745} C_VEL
LIN {X 0,Y 245.524,Z 813.45,A -85,B 0,C 180,E1 -19150.628,E2 -19150.628} C_VEL
LIN {X 0,Y 244.222,Z 821.337,A -85,B 0,C 180,E1 -19152.412,E2 -19152.412} C_VEL
LIN {X 0,Y 242.613,Z 830.238,A -85,B 0,C 180,E1 -19154.887,E2 -19154.887} C_VEL
LIN {X 0,Y 241.342,Z 837.368,A -85,B 0,C 180,E1 -19157.384,E2 -19157.384} C_VEL
LIN {X 0,Y 240.616,Z 843.028,A -85,B 0,C 180,E1 -19159.906,E2 -19159.906} C_VEL
LIN {X 0,Y 240.151,Z 847.44,A -85,B 0,C 180,E1 -19162.432,E2 -19162.432} C_VEL
LIN {X 0,Y 239.922,Z 850.73,A -85,B 0,C 180,E1 -19164.958,E2 -19164.958} C_VEL
LIN {X 0,Y 239.912,Z 852.345,A -85,B 0,C 180,E1 -19166.64,E2 -19166.64} C_VEL
LIN {X 0,Y 239.982,Z 853.541,A -85,B 0,C 180,E1 -19168.321,E2 -19168.321} C_VEL
LIN {X 0,Y 239.996,Z 854.277,A -85,B 0,C 180,E1 -19169.999,E2 -19169.999} C_VEL
LIN {X 0,Y 239.945,Z 854.593,A -85,B 0,C 180,E1 -19171.678,E2 -19171.678} C_VEL
LIN {X 0,Y 239.854,Z 854.514,A -85,B 0,C 180,E1 -19173.359,E2 -19173.359} C_VEL
LIN {X 0,Y 239.881,Z 854.041,A -85,B 0,C 180,E1 -19175.041,E2 -19175.041} C_VEL
LIN {X 0,Y 240.028,Z 853.13,A -85,B 0,C 180,E1 -19176.725,E2 -19176.725} C_VEL
LIN {X 0,Y 240.748,Z 850.104,A -85,B 0,C 180,E1 -19180.087,E2 -19180.087} C_VEL
LIN {X 0,Y 241.677,Z 846.694,A -85,B 0,C 180,E1 -19182.597,E2 -19182.597} C_VEL
LIN {X 0,Y 242.998,Z 842.246,A -85,B 0,C 180,E1 -19185.087,E2 -19185.087} C_VEL
LIN {X 0,Y 245.345,Z 835.548,A -85,B 0,C 180,E1 -19187.934,E2 -19187.934} C_VEL
LIN {X 0,Y 247.717,Z 827.617,A -85,B 0,C 180,E1 -19190.568,E2 -19190.568} C_VEL
LIN {X 0,Y 250.318,Z 819.443,A -85,B 0,C 180,E1 -19192.708,E2 -19192.708} C_VEL
LIN {X 0,Y 253.002,Z 810.33,A -85,B 0,C 180,E1 -19194.624,E2 -19194.624} C_VEL
LIN {X 0,Y 256.017,Z 799.197,A -85,B 0,C 180,E1 -19196.491,E2 -19196.491} C_VEL
LIN {X 0,Y 257.671,Z 788.048,A -85,B 0,C 180,E1 -19198.119,E2 -19198.119} C_VEL
LIN {X 0,Y 258.906,Z 776.091,A -85,B 0,C 180,E1 -19199.527,E2 -19199.527} C_VEL
LIN {X 0,Y 258.622,Z 764.549,A -85,B 0,C 180,E1 -19200.801,E2 -19200.801} C_VEL
LIN {X 0,Y 256.946,Z 751.783,A -85,B 0,C 180,E1 -19202.152,E2 -19202.152} C_VEL
LIN {X 0,Y 253.409,Z 737.062,A -85,B 0,C 180,E1 -19203.741,E2 -19203.741} C_VEL
LIN {X 0,Y 253.675,Z 725.567,A -85,B 0,C 180,E1 -19206.54,E2 -19206.54} C_VEL
LIN {X 0,Y 254.12,Z 715.015,A -85,B 0,C 180,E1 -19209.5,E2 -19209.5} C_VEL
LIN {X 0,Y 254.312,Z 709.962,A -85,B 0,C 180,E1 -19211.144,E2 -19211.144} C_VEL
LIN {X 0,Y 252.984,Z 702.976,A -85,B 0,C 180,E1 -19214.385,E2 -19214.385} C_VEL
LIN {X 0,Y 252.111,Z 696.747,A -85,B 0,C 180,E1 -19218.007,E2 -19218.007} C_VEL
LIN {X 0,Y 252.027,Z 692.158,A -85,B 0,C 180,E1 -19221.332,E2 -19221.332} C_VEL
LIN {X 0,Y 251.782,Z 691.391,A -85,B 0,C 180,E1 -19222.114,E2 -19222.114} C_VEL
LIN {X 0,Y 251.167,Z 690.085,A -85,B 0,C 180,E1 -19224.237,E2 -19224.237} C_VEL
LIN {X 0,Y 250.231,Z 688.756,A -85,B 0,C 180,E1 -19227.748,E2 -19227.748} C_VEL
LIN {X 0,Y 249.976,Z 688.452,A -85,B 0,C 180,E1 -19231.448,E2 -19231.448} C_VEL
LIN {X 0,Y 250.169,Z 689.073,A -85,B 0,C 180,E1 -19235.077,E2 -19235.077} C_VEL
LIN {X 0,Y 250.545,Z 690.823,A -85,B 0,C 180,E1 -19238.613,E2 -19238.613} C_VEL
LIN {X 0,Y 251.104,Z 692.979,A -85,B 0,C 180,E1 -19242.098,E2 -19242.098} C_VEL
LIN {X 0,Y 251.899,Z 696.054,A -85,B 0,C 180,E1 -19245.457,E2 -19245.457} C_VEL
LIN {X 0,Y 253.068,Z 700.78,A -85,B 0,C 180,E1 -19249.6,E2 -19249.6} C_VEL
LIN {X 0,Y 253.74,Z 704.005,A -85,B 0,C 180,E1 -19252.039,E2 -19252.039} C_VEL
LIN {X 0,Y 254.525,Z 709.848,A -85,B 0,C 180,E1 -19255.846,E2 -19255.846} C_VEL
LIN {X 0,Y 254.746,Z 714.325,A -85,B 0,C 180,E1 -19258.419,E2 -19258.419} C_VEL
LIN {X 0,Y 254.175,Z 719.105,A -85,B 0,C 180,E1 -19260.792,E2 -19260.792} C_VEL
LIN {X 0,Y 252.093,Z 728.297,A -85,B 0,C 180,E1 -19264.936,E2 -19264.936} C_VEL
LIN {X 0,Y 251.233,Z 732.721,A -85,B 0,C 180,E1 -19266.878,E2 -19266.878} C_VEL
LIN {X 0,Y 255.612,Z 746.507,A -85,B 0,C 180,E1 -19268.747,E2 -19268.747} C_VEL
LIN {X 0,Y 258.071,Z 758.218,A -85,B 0,C 180,E1 -19270.343,E2 -19270.343} C_VEL
LIN {X 0,Y 259.367,Z 770.697,A -85,B 0,C 180,E1 -19272.122,E2 -19272.122} C_VEL
LIN {X 0,Y 259.45,Z 778.582,A -85,B 0,C 180,E1 -19273.311,E2 -19273.311} C_VEL
LIN {X 0,Y 256.816,Z 789.643,A -85,B 0,C 180,E1 -19274.866,E2 -19274.866} C_VEL
LIN {X 0,Y 254.044,Z 799.891,A -85,B 0,C 180,E1 -19276.679,E2 -19276.679} C_VEL
LIN {X 0,Y 251.448,Z 808.399,A -85,B 0,C 180,E1 -19278.551,E2 -19278.551} C_VEL
LIN {X 0,Y 248.517,Z 817.461,A -85,B 0,C 180,E1 -19281.059,E2 -19281.059} C_VEL
LIN {X 0,Y 246.099,Z 824.568,A -85,B 0,C 180,E1 -19283.566,E2 -19283.566} C_VEL
LIN {X 0,Y 244.066,Z 830.133,A -85,B 0,C 180,E1 -19286.082,E2 -19286.082} C_VEL
LIN {X 0,Y 242.622,Z 834.252,A -85,B 0,C 180,E1 -19288.491,E2 -19288.491} C_VEL
LIN {X 0,Y 241.206,Z 838.12,A -85,B 0,C 180,E1 -19291.632,E2 -19291.632} C_VEL
LIN {X 0,Y 240.13,Z 840.594,A -85,B 0,C 180,E1 -19294.969,E2 -19294.969} C_VEL
LIN {X 0,Y 239.599,Z 841.433,A -85,B 0,C 180,E1 -19298.023,E2 -19298.023} C_VEL
LIN {X 0,Y 239.418,Z 841.229,A -85,B 0,C 180,E1 -19300.253,E2 -19300.253} C_VEL
LIN {X 0,Y 239.392,Z 840.134,A -85,B 0,C 180,E1 -19302.784,E2 -19302.784} C_VEL
LIN {X 0,Y 239.745,Z 837.249,A -85,B 0,C 180,E1 -19306.105,E2 -19306.105} C_VEL
LIN {X 0,Y 240.275,Z 833.896,A -85,B 0,C 180,E1 -19308.638,E2 -19308.638} C_VEL
LIN {X 0,Y 240.859,Z 829.763,A -85,B 0,C 180,E1 -19311.002,E2 -19311.002} C_VEL
LIN {X 0,Y 242.05,Z 823.162,A -85,B 0,C 180,E1 -19313.914,E2 -19313.914} C_VEL
LIN {X 0,Y 243.203,Z 816.555,A -85,B 0,C 180,E1 -19316.202,E2 -19316.202} C_VEL
LIN {X 0,Y 244.856,Z 807.743,A -85,B 0,C 180,E1 -19318.653,E2 -19318.653} C_VEL
LIN {X 0,Y 246.616,Z 798.136,A -85,B 0,C 180,E1 -19320.79,E2 -19320.79} C_VEL
LIN {X 0,Y 248.372,Z 787.841,A -85,B 0,C 180,E1 -19322.626,E2 -19322.626} C_VEL
LIN {X 0,Y 250.075,Z 776.56,A -85,B 0,C 180,E1 -19324.239,E2 -19324.239} C_VEL
LIN {X 0,Y 250.848,Z 770.923,A -85,B 0,C 180,E1 -19324.907,E2 -19324.907} C_VEL
LIN {X 0,Y 249.742,Z 760.055,A -85,B 0,C 180,E1 -19326.171,E2 -19326.171} C_VEL
LIN {X 0,Y 247.964,Z 746.572,A -85,B 0,C 180,E1 -19327.424,E2 -19327.424} C_VEL
LIN {X 0,Y 245.511,Z 733.053,A -85,B 0,C 180,E1 -19328.374,E2 -19328.374} C_VEL
LIN {X 0,Y 245.19,Z 731.187,A -85,B 0,C 180,E1 -19328.51,E2 -19328.51} C_VEL
LIN {X 0,Y 246.188,Z 722.281,A -85,B 0,C 180,E1 -19332.13,E2 -19332.13} C_VEL
LIN {X 0,Y 247.303,Z 712.664,A -85,B 0,C 180,E1 -19336.079,E2 -19336.079} C_VEL
LIN {X 0,Y 248.205,Z 704.604,A -85,B 0,C 180,E1 -19339.395,E2 -19339.395} C_VEL
LIN {X 0,Y 248.318,Z 700.714,A -85,B 0,C 180,E1 -19341.046,E2 -19341.046} C_VEL
LIN {X 0,Y 247.683,Z 695.258,A -85,B 0,C 180,E1 -19343.484,E2 -19343.484} C_VEL
LIN {X 0,Y 245.828,Z 684.823,A -85,B 0,C 180,E1 -19348.363,E2 -19348.363} C_VEL
LIN {X 0,Y 244.892,Z 679.653,A -85,B 0,C 180,E1 -19350.823,E2 -19350.823} C_VEL
LIN {X 0,Y 242.987,Z 673.128,A -85,B 0,C 180,E1 -19354.147,E2 -19354.147} C_VEL
LIN {X 0,Y 242.306,Z 670.301,A -85,B 0,C 180,E1 -19355.619,E2 -19355.619} C_VEL
LIN {X 0,Y 242.426,Z 670.289,A -85,B 0,C 180,E1 -19358.335,E2 -19358.335} C_VEL
LIN {X 0,Y 242.241,Z 670.31,A -85,B 0,C 180,E1 -19361.188,E2 -19361.188} C_VEL
LIN {X 0,Y 246.688,Z 683.103,A -85,B 0,C 180,E1 -19362.945,E2 -19362.945} C_VEL
LIN {X 0,Y 249.925,Z 693.931,A -85,B 0,C 180,E1 -19364.661,E2 -19364.661} C_VEL
LIN {X 0,Y 251.805,Z 701.269,A -85,B 0,C 180,E1 -19365.98,E2 -19365.98} C_VEL
LIN {X 0,Y 251.746,Z 703.844,A -85,B 0,C 180,E1 -19366.407,E2 -19366.407} C_VEL
LIN {X 0,Y 249.979,Z 714.982,A -85,B 0,C 180,E1 -19368.439,E2 -19368.439} C_VEL
LIN {X 0,Y 248.295,Z 724.879,A -85,B 0,C 180,E1 -19370.703,E2 -19370.703} C_VEL
LIN {X 0,Y 246.713,Z 733.108,A -85,B 0,C 180,E1 -19373.06,E2 -19373.06} C_VEL
LIN {X 0,Y 245.234,Z 740.848,A -85,B 0,C 180,E1 -19375.851,E2 -19375.851} C_VEL
LIN {X 0,Y 244.24,Z 746.252,A -85,B 0,C 180,E1 -19378.346,E2 -19378.346} C_VEL
LIN {X 0,Y 243.368,Z 751.12,A -85,B 0,C 180,E1 -19381.32,E2 -19381.32} C_VEL
LIN {X 0,Y 242.927,Z 753.64,A -85,B 0,C 180,E1 -19383.346,E2 -19383.346} C_VEL
LIN {X 0,Y 242.626,Z 755.811,A -85,B 0,C 180,E1 -19385.801,E2 -19385.801} C_VEL
LIN {X 0,Y 242.691,Z 757.203,A -85,B 0,C 180,E1 -19388.567,E2 -19388.567} C_VEL
LIN {X 0,Y 243.182,Z 757.44,A -85,B 0,C 180,E1 -19391.66,E2 -19391.66} C_VEL
LIN {X 0,Y 243.799,Z 756.805,A -85,B 0,C 180,E1 -19393.89,E2 -19393.89} C_VEL
LIN {X 0,Y 244.775,Z 755.159,A -85,B 0,C 180,E1 -19396.442,E2 -19396.442} C_VEL
LIN {X 0,Y 246.051,Z 752.574,A -85,B 0,C 180,E1 -19398.932,E2 -19398.932} C_VEL
LIN {X 0,Y 247.502,Z 749.084,A -85,B 0,C 180,E1 -19401.34,E2 -19401.34} C_VEL
LIN {X 0,Y 249.582,Z 743.769,A -85,B 0,C 180,E1 -19404.054,E2 -19404.054} C_VEL
LIN {X 0,Y 252.048,Z 736.727,A -85,B 0,C 180,E1 -19406.774,E2 -19406.774} C_VEL
LIN {X 0,Y 254.515,Z 728.79,A -85,B 0,C 180,E1 -19409.161,E2 -19409.161} C_VEL
LIN {X 0,Y 257.162,Z 719.534,A -85,B 0,C 180,E1 -19411.324,E2 -19411.324} C_VEL
LIN {X 0,Y 258.667,Z 713.602,A -85,B 0,C 180,E1 -19412.491,E2 -19412.491} C_VEL
LIN {X 0,Y 258.327,Z 709.997,A -85,B 0,C 180,E1 -19413.327,E2 -19413.327} C_VEL
LIN {X 0,Y 256.288,Z 701.721,A -85,B 0,C 180,E1 -19415.279,E2 -19415.279} C_VEL
LIN {X 0,Y 252.772,Z 691.837,A -85,B 0,C 180,E1 -19417.524,E2 -19417.524} C_VEL
LIN {X 0,Y 248.279,Z 682.058,A -85,B 0,C 180,E1 -19419.711,E2 -19419.711} C_VEL
LIN {X 0,Y 246.634,Z 678.719,A -85,B 0,C 180,E1 -19420.438,E2 -19420.438} C_VEL
LIN {X 0,Y 244.798,Z 675.652,A -85,B 0,C 180,E1 -19421.156,E2 -19421.156} C_VEL
LIN {X 0,Y 243.736,Z 674.02,A -85,B 0,C 180,E1 -19421.562,E2 -19421.562} C_VEL
LIN {X 0,Y 242.346,Z 671.47,A -85,B 0,C 180,E1 -19422.109,E2 -19422.109} C_VEL
LIN {X 0,Y 242.098,Z 670.33,A -85,B 0,C 180,E1 -19422.308,E2 -19422.308} C_VEL
LIN {X 0,Y 242.169,Z 670.319,A -85,B 0,C 180,E1 -19426.575,E2 -19426.575} C_VEL
LIN {X 0,Y 242.43,Z 670.277,A -85,B 0,C 180,E1 -19431.666,E2 -19431.666} C_VEL
LIN {X 0,Y 242.264,Z 670.307,A -85,B 0,C 180,E1 -19435.008,E2 -19435.008} C_VEL
LIN {X 0,Y 242.639,Z 670.258,A -85,B 0,C 180,E1 -19438.34,E2 -19438.34} C_VEL
LIN {X 0,Y 242.64,Z 670.249,A -85,B 0,C 180,E1 -19441.66,E2 -19441.66} C_VEL
LIN {X 0,Y 242.436,Z 670.284,A -85,B 0,C 180,E1 -19446.659,E2 -19446.659} C_VEL
LIN {X 0,Y 242.317,Z 670.293,A -85,B 0,C 180,E1 -19450.022,E2 -19450.022} C_VEL
LIN {X 0,Y 242.17,Z 670.319,A -85,B 0,C 180,E1 -19455.141,E2 -19455.141} C_VEL
LIN {X 0,Y 242.076,Z 670.33,A -85,B 0,C 180,E1 -19458.624,E2 -19458.624} C_VEL
LIN {X 0,Y 242.029,Z 670.328,A -85,B 0,C 180,E1 -19460.008,E2 -19460.008} C_VEL
LIN {X 0,Y 241.355,Z 670.421,A -85,B 0,C 180,E1 -19461.399,E2 -19461.399} C_VEL
LIN {X 0,Y 238.437,Z 670.779,A -85,B 0,C 180,E1 -19463.668,E2 -19463.668} C_VEL
LIN {X 0,Y 236.056,Z 671.246,A -85,B 0,C 180,E1 -19465.509,E2 -19465.509} C_VEL
LIN {X 0,Y 235.172,Z 671.956,A -85,B 0,C 180,E1 -19466.928,E2 -19466.928} C_VEL
LIN {X 0,Y 235.174,Z 672.307,A -85,B 0,C 180,E1 -19467.403,E2 -19467.403} C_VEL
LIN {X 0,Y 235.784,Z 674.957,A -85,B 0,C 180,E1 -19470.446,E2 -19470.446} C_VEL
LIN {X 0,Y 236.923,Z 679.924,A -85,B 0,C 180,E1 -19475.341,E2 -19475.341} C_VEL
LIN {X 0,Y 237.684,Z 683.416,A -85,B 0,C 180,E1 -19478.385,E2 -19478.385} C_VEL
LIN {X 0,Y 238.719,Z 688.883,A -85,B 0,C 180,E1 -19482.62,E2 -19482.62} C_VEL
LIN {X 0,Y 239.614,Z 693.691,A -85,B 0,C 180,E1 -19486.02,E2 -19486.02} C_VEL
LIN {X 0,Y 240.431,Z 699.001,A -85,B 0,C 180,E1 -19489.465,E2 -19489.465} C_VEL
LIN {X 0,Y 240.301,Z 701.684,A -85,B 0,C 180,E1 -19491.037,E2 -19491.037} C_VEL
LIN {X 0,Y 238.774,Z 707.696,A -85,B 0,C 180,E1 -19494.309,E2 -19494.309} C_VEL
LIN {X 0,Y 239.751,Z 711.74,A -85,B 0,C 180,E1 -19494.752,E2 -19494.752} C_VEL
LIN {X 0,Y 242.218,Z 722.517,A -85,B 0,C 180,E1 -19496.059,E2 -19496.059} C_VEL
LIN {X 0,Y 244.191,Z 733.84,A -85,B 0,C 180,E1 -19497.496,E2 -19497.496} C_VEL
LIN {X 0,Y 245.229,Z 746.431,A -85,B 0,C 180,E1 -19499.178,E2 -19499.178} C_VEL
LIN {X 0,Y 245.251,Z 759.153,A -85,B 0,C 180,E1 -19501.08,E2 -19501.08} C_VEL
LIN {X 0,Y 244.45,Z 769.675,A -85,B 0,C 180,E1 -19502.858,E2 -19502.858} C_VEL
LIN {X 0,Y 242.991,Z 779.416,A -85,B 0,C 180,E1 -19504.747,E2 -19504.747} C_VEL
LIN {X 0,Y 242.489,Z 782.964,A -85,B 0,C 180,E1 -19505.492,E2 -19505.492} C_VEL
LIN {X 0,Y 241.91,Z 793.915,A -85,B 0,C 180,E1 -19506.908,E2 -19506.908} C_VEL
LIN {X 0,Y 240.141,Z 804.396,A -85,B 0,C 180,E1 -19508.541,E2 -19508.541} C_VEL
LIN {X 0,Y 238.44,Z 814.36,A -85,B 0,C 180,E1 -19510.488,E2 -19510.488} C_VEL
LIN {X 0,Y 237.117,Z 822.061,A -85,B 0,C 180,E1 -19512.324,E2 -19512.324} C_VEL
LIN {X 0,Y 235.457,Z 830.76,A -85,B 0,C 180,E1 -19514.86,E2 -19514.86} C_VEL
LIN {X 0,Y 234.223,Z 837.709,A -85,B 0,C 180,E1 -19517.435,E2 -19517.435} C_VEL
LIN {X 0,Y 233.403,Z 844.065,A -85,B 0,C 180,E1 -19520.466,E2 -19520.466} C_VEL
LIN {X 0,Y 233.004,Z 848.184,A -85,B 0,C 180,E1 -19523.069,E2 -19523.069} C_VEL
LIN {X 0,Y 232.843,Z 850.42,A -85,B 0,C 180,E1 -19524.91,E2 -19524.91} C_VEL
LIN {X 0,Y 232.888,Z 853.201,A -85,B 0,C 180,E1 -19528.27,E2 -19528.27} C_VEL
LIN {X 0,Y 232.925,Z 854.013,A -85,B 0,C 180,E1 -19529.999,E2 -19529.999} C_VEL
LIN {X 0,Y 232.851,Z 854.37,A -85,B 0,C 180,E1 -19531.729,E2 -19531.729} C_VEL
LIN {X 0,Y 232.801,Z 853.898,A -85,B 0,C 180,E1 -19535.195,E2 -19535.195} C_VEL
LIN {X 0,Y 232.948,Z 853.058,A -85,B 0,C 180,E1 -19536.93,E2 -19536.93} C_VEL
LIN {X 0,Y 233.739,Z 850.123,A -85,B 0,C 180,E1 -19540.392,E2 -19540.392} C_VEL
LIN {X 0,Y 234.736,Z 846.818,A -85,B 0,C 180,E1 -19542.975,E2 -19542.975} C_VEL
LIN {X 0,Y 236.156,Z 842.469,A -85,B 0,C 180,E1 -19545.535,E2 -19545.535} C_VEL
LIN {X 0,Y 238.613,Z 835.929,A -85,B 0,C 180,E1 -19548.458,E2 -19548.458} C_VEL
LIN {X 0,Y 241.001,Z 828.446,A -85,B 0,C 180,E1 -19551.064,E2 -19551.064} C_VEL
LIN {X 0,Y 243.834,Z 820.156,A -85,B 0,C 180,E1 -19553.347,E2 -19553.347} C_VEL
LIN {X 0,Y 246.627,Z 811.334,A -85,B 0,C 180,E1 -19555.305,E2 -19555.305} C_VEL
LIN {X 0,Y 249.791,Z 800.466,A -85,B 0,C 180,E1 -19557.205,E2 -19557.205} C_VEL
LIN {X 0,Y 251.633,Z 789.318,A -85,B 0,C 180,E1 -19558.909,E2 -19558.909} C_VEL
LIN {X 0,Y 253.128,Z 776.904,A -85,B 0,C 180,E1 -19560.453,E2 -19560.453} C_VEL
LIN {X 0,Y 253.06,Z 766.812,A -85,B 0,C 180,E1 -19561.645,E2 -19561.645} C_VEL
LIN {X 0,Y 251.603,Z 754.129,A -85,B 0,C 180,E1 -19563.071,E2 -19563.071} C_VEL
LIN {X 0,Y 248.349,Z 739.85,A -85,B 0,C 180,E1 -19564.704,E2 -19564.704} C_VEL
LIN {X 0,Y 247.641,Z 736.763,A -85,B 0,C 180,E1 -19565.125,E2 -19565.125} C_VEL
LIN {X 0,Y 248.109,Z 725.74,A -85,B 0,C 180,E1 -19568.017,E2 -19568.017} C_VEL
LIN {X 0,Y 248.737,Z 717.241,A -85,B 0,C 180,E1 -19570.529,E2 -19570.529} C_VEL
LIN {X 0,Y 248.85,Z 713.924,A -85,B 0,C 180,E1 -19571.665,E2 -19571.665} C_VEL
LIN {X 0,Y 247.686,Z 707.321,A -85,B 0,C 180,E1 -19574.816,E2 -19574.816} C_VEL
LIN {X 0,Y 246.97,Z 702.291,A -85,B 0,C 180,E1 -19577.719,E2 -19577.719} C_VEL
LIN {X 0,Y 246.832,Z 697.392,A -85,B 0,C 180,E1 -19581.214,E2 -19581.214} C_VEL
LIN {X 0,Y 246.301,Z 695.629,A -85,B 0,C 180,E1 -19583.186,E2 -19583.186} C_VEL
LIN {X 0,Y 245.477,Z 694.143,A -85,B 0,C 180,E1 -19586.124,E2 -19586.124} C_VEL
LIN {X 0,Y 244.711,Z 693.159,A -85,B 0,C 180,E1 -19590.775,E2 -19590.775} C_VEL
LIN {X 0,Y 244.744,Z 693.55,A -85,B 0,C 180,E1 -19594.485,E2 -19594.485} C_VEL
LIN {X 0,Y 244.964,Z 695.032,A -85,B 0,C 180,E1 -19598.101,E2 -19598.101} C_VEL
LIN {X 0,Y 245.459,Z 697.097,A -85,B 0,C 180,E1 -19601.642,E2 -19601.642} C_VEL
LIN {X 0,Y 246.108,Z 699.995,A -85,B 0,C 180,E1 -19605.107,E2 -19605.107} C_VEL
LIN {X 0,Y 247.12,Z 704.504,A -85,B 0,C 180,E1 -19609.347,E2 -19609.347} C_VEL
LIN {X 0,Y 247.754,Z 707.708,A -85,B 0,C 180,E1 -19611.846,E2 -19611.846} C_VEL
LIN {X 0,Y 248.404,Z 713.782,A -85,B 0,C 180,E1 -19615.944,E2 -19615.944} C_VEL
LIN {X 0,Y 248.462,Z 717.931,A -85,B 0,C 180,E1 -19618.379,E2 -19618.379} C_VEL
LIN {X 0,Y 247.677,Z 722.767,A -85,B 0,C 180,E1 -19620.813,E2 -19620.813} C_VEL
LIN {X 0,Y 245.259,Z 732.809,A -85,B 0,C 180,E1 -19625.441,E2 -19625.441} C_VEL
LIN {X 0,Y 249.561,Z 746.343,A -85,B 0,C 180,E1 -19627.433,E2 -19627.433} C_VEL
LIN {X 0,Y 251.927,Z 757.374,A -85,B 0,C 180,E1 -19629.028,E2 -19629.028} C_VEL
LIN {X 0,Y 253.22,Z 767.526,A -85,B 0,C 180,E1 -19630.543,E2 -19630.543} C_VEL
LIN {X 0,Y 253.592,Z 777.995,A -85,B 0,C 180,E1 -19632.199,E2 -19632.199} C_VEL
LIN {X 0,Y 253.144,Z 781.516,A -85,B 0,C 180,E1 -19632.723,E2 -19632.723} C_VEL
LIN {X 0,Y 250.221,Z 792.708,A -85,B 0,C 180,E1 -19634.414,E2 -19634.414} C_VEL
LIN {X 0,Y 246.897,Z 803.7,A -85,B 0,C 180,E1 -19636.538,E2 -19636.538} C_VEL
LIN {X 0,Y 244.321,Z 811.536,A -85,B 0,C 180,E1 -19638.446,E2 -19638.446} C_VEL
LIN {X 0,Y 241.598,Z 819.256,A -85,B 0,C 180,E1 -19640.782,E2 -19640.782} C_VEL
LIN {X 0,Y 239.245,Z 825.64,A -85,B 0,C 180,E1 -19643.204,E2 -19643.204} C_VEL
LIN {X 0,Y 237.41,Z 830.355,A -85,B 0,C 180,E1 -19645.419,E2 -19645.419} C_VEL
LIN {X 0,Y 235.496,Z 835.351,A -85,B 0,C 180,E1 -19648.522,E2 -19648.522} C_VEL
LIN {X 0,Y 234.497,Z 837.851,A -85,B 0,C 180,E1 -19650.63,E2 -19650.63} C_VEL
LIN {X 0,Y 233.71,Z 839.734,A -85,B 0,C 180,E1 -19652.771,E2 -19652.771} C_VEL
LIN {X 0,Y 232.925,Z 841.182,A -85,B 0,C 180,E1 -19655.448,E2 -19655.448} C_VEL
LIN {X 0,Y 232.475,Z 841.673,A -85,B 0,C 180,E1 -19658.188,E2 -19658.188} C_VEL
LIN {X 0,Y 232.276,Z 841.185,A -85,B 0,C 180,E1 -19660.852,E2 -19660.852} C_VEL
LIN {X 0,Y 232.375,Z 839.319,A -85,B 0,C 180,E1 -19664.076,E2 -19664.076} C_VEL
LIN {X 0,Y 232.899,Z 835.785,A -85,B 0,C 180,E1 -19667.45,E2 -19667.45} C_VEL
LIN {X 0,Y 233.438,Z 832.177,A -85,B 0,C 180,E1 -19669.864,E2 -19669.864} C_VEL
LIN {X 0,Y 234.426,Z 826.564,A -85,B 0,C 180,E1 -19672.745,E2 -19672.745} C_VEL
LIN {X 0,Y 235.673,Z 819.6,A -85,B 0,C 180,E1 -19675.488,E2 -19675.488} C_VEL
LIN {X 0,Y 237.316,Z 811.261,A -85,B 0,C 180,E1 -19678.088,E2 -19678.088} C_VEL
LIN {X 0,Y 238.986,Z 802.098,A -85,B 0,C 180,E1 -19680.366,E2 -19680.366} C_VEL
LIN {X 0,Y 240.859,Z 791.962,A -85,B 0,C 180,E1 -19682.385,E2 -19682.385} C_VEL
LIN {X 0,Y 242.585,Z 781.455,A -85,B 0,C 180,E1 -19684.075,E2 -19684.075} C_VEL
LIN {X 0,Y 243.993,Z 771.859,A -85,B 0,C 180,E1 -19685.314,E2 -19685.314} C_VEL
LIN {X 0,Y 243.022,Z 761.529,A -85,B 0,C 180,E1 -19686.57,E2 -19686.57} C_VEL
LIN {X 0,Y 241.337,Z 748.238,A -85,B 0,C 180,E1 -19687.868,E2 -19687.868} C_VEL
LIN {X 0,Y 238.989,Z 734.805,A -85,B 0,C 180,E1 -19688.886,E2 -19688.886} C_VEL
LIN {X 0,Y 238.337,Z 731.358,A -85,B 0,C 180,E1 -19689.109,E2 -19689.109} C_VEL
LIN {X 0,Y 239.298,Z 723.242,A -85,B 0,C 180,E1 -19692.481,E2 -19692.481} C_VEL
LIN {X 0,Y 240.458,Z 713.664,A -85,B 0,C 180,E1 -19696.479,E2 -19696.479} C_VEL
LIN {X 0,Y 241.418,Z 705.412,A -85,B 0,C 180,E1 -19699.942,E2 -19699.942} C_VEL
LIN {X 0,Y 241.346,Z 700.924,A -85,B 0,C 180,E1 -19701.923,E2 -19701.923} C_VEL
LIN {X 0,Y 240.401,Z 694.367,A -85,B 0,C 180,E1 -19704.969,E2 -19704.969} C_VEL
LIN {X 0,Y 238.615,Z 683.856,A -85,B 0,C 180,E1 -19710.001,E2 -19710.001} C_VEL
LIN {X 0,Y 237.387,Z 678.842,A -85,B 0,C 180,E1 -19712.546,E2 -19712.546} C_VEL
LIN {X 0,Y 235.396,Z 671.157,A -85,B 0,C 180,E1 -19716.644,E2 -19716.644} C_VEL
LIN {X 0,Y 235.269,Z 671.337,A -85,B 0,C 180,E1 -19720.543,E2 -19720.543} C_VEL
LIN {X 0,Y 239.58,Z 683.711,A -85,B 0,C 180,E1 -19722.276,E2 -19722.276} C_VEL
LIN {X 0,Y 242.886,Z 694.562,A -85,B 0,C 180,E1 -19724.057,E2 -19724.057} C_VEL
LIN {X 0,Y 245.031,Z 702.838,A -85,B 0,C 180,E1 -19725.599,E2 -19725.599} C_VEL
LIN {X 0,Y 244.725,Z 706.674,A -85,B 0,C 180,E1 -19726.261,E2 -19726.261} C_VEL
LIN {X 0,Y 242.944,Z 717.354,A -85,B 0,C 180,E1 -19728.316,E2 -19728.316} C_VEL
LIN {X 0,Y 241.347,Z 726.253,A -85,B 0,C 180,E1 -19730.454,E2 -19730.454} C_VEL
LIN {X 0,Y 239.755,Z 734.316,A -85,B 0,C 180,E1 -19732.843,E2 -19732.843} C_VEL
LIN {X 0,Y 238.42,Z 741.023,A -85,B 0,C 180,E1 -19735.305,E2 -19735.305} C_VEL
LIN {X 0,Y 237.523,Z 745.71,A -85,B 0,C 180,E1 -19737.42,E2 -19737.42} C_VEL
LIN {X 0,Y 236.552,Z 751.075,A -85,B 0,C 180,E1 -19740.504,E2 -19740.504} C_VEL
LIN {X 0,Y 235.859,Z 754.77,A -85,B 0,C 180,E1 -19743.454,E2 -19743.454} C_VEL
LIN {X 0,Y 235.589,Z 757.299,A -85,B 0,C 180,E1 -19746.63,E2 -19746.63} C_VEL
LIN {X 0,Y 235.731,Z 758.347,A -85,B 0,C 180,E1 -19749.181,E2 -19749.181} C_VEL
LIN {X 0,Y 236.221,Z 758.495,A -85,B 0,C 180,E1 -19751.945,E2 -19751.945} C_VEL
LIN {X 0,Y 237.288,Z 757.301,A -85,B 0,C 180,E1 -19755.303,E2 -19755.303} C_VEL
LIN {X 0,Y 238.871,Z 754.538,A -85,B 0,C 180,E1 -19758.613,E2 -19758.613} C_VEL
LIN {X 0,Y 240.182,Z 751.758,A -85,B 0,C 180,E1 -19760.843,E2 -19760.843} C_VEL
LIN {X 0,Y 242.191,Z 746.934,A -85,B 0,C 180,E1 -19763.668,E2 -19763.668} C_VEL
LIN {X 0,Y 244.634,Z 740.652,A -85,B 0,C 180,E1 -19766.422,E2 -19766.422} C_VEL
LIN {X 0,Y 246.921,Z 734.205,A -85,B 0,C 180,E1 -19768.637,E2 -19768.637} C_VEL
LIN {X 0,Y 249.47,Z 726.188,A -85,B 0,C 180,E1 -19770.848,E2 -19770.848} C_VEL
LIN {X 0,Y 252.068,Z 717.009,A -85,B 0,C 180,E1 -19772.858,E2 -19772.858} C_VEL
LIN {X 0,Y 252.461,Z 714.873,A -85,B 0,C 180,E1 -19773.305,E2 -19773.305} C_VEL
LIN {X 0,Y 250.74,Z 706.266,A -85,B 0,C 180,E1 -19775.47,E2 -19775.47} C_VEL
LIN {X 0,Y 247.506,Z 696.305,A -85,B 0,C 180,E1 -19777.899,E2 -19777.899} C_VEL
LIN {X 0,Y 243.421,Z 686.826,A -85,B 0,C 180,E1 -19780.169,E2 -19780.169} C_VEL
LIN {X 0,Y 240.271,Z 680.697,A -85,B 0,C 180,E1 -19781.673,E2 -19781.673} C_VEL
LIN {X 0,Y 237.694,Z 676.041,A -85,B 0,C 180,E1 -19782.802,E2 -19782.802} C_VEL
LIN {X 0,Y 235.619,Z 673.06,A -85,B 0,C 180,E1 -19783.606,E2 -19783.606} C_VEL
LIN {X 0,Y 235.106,Z 671.203,A -85,B 0,C 180,E1 -19783.982,E2 -19783.982} C_VEL
LIN {X 0,Y 235.149,Z 671.191,A -85,B 0,C 180,E1 -19787.924,E2 -19787.924} C_VEL
LIN {X 0,Y 235.38,Z 671.158,A -85,B 0,C 180,E1 -19791.414,E2 -19791.414} C_VEL
LIN {X 0,Y 235.407,Z 671.151,A -85,B 0,C 180,E1 -19793.142,E2 -19793.142} C_VEL
LIN {X 0,Y 235.599,Z 671.134,A -85,B 0,C 180,E1 -19798.291,E2 -19798.291} C_VEL
LIN {X 0,Y 235.599,Z 671.126,A -85,B 0,C 180,E1 -19801.71,E2 -19801.71} C_VEL
LIN {X 0,Y 235.407,Z 671.162,A -85,B 0,C 180,E1 -19806.859,E2 -19806.859} C_VEL
LIN {X 0,Y 235.241,Z 671.177,A -85,B 0,C 180,E1 -19810.327,E2 -19810.327} C_VEL
LIN {X 0,Y 235.117,Z 671.193,A -85,B 0,C 180,E1 -19815.606,E2 -19815.606} C_VEL
LIN {X 0,Y 234.984,Z 671.206,A -85,B 0,C 180,E1 -19820.005,E2 -19820.005} C_VEL
LIN {X 0,Y 234.964,Z 671.21,A -85,B 0,C 180,E1 -19822.883,E2 -19822.883} C_VEL
LIN {X 0,Y 235.022,Z 671.334,A -85,B 0,C 180,E1 -19826.218,E2 -19826.218} C_VEL
LIN {X 0,Y 235.174,Z 672.307,A -85,B 0,C 180,E1 -19827.403,E2 -19827.403} C_VEL
LIN {X 0,Y 234.818,Z 673.698,A -85,B 0,C 180,E1 -19828.796,E2 -19828.796} C_VEL
LIN {X 0,Y 232.544,Z 676.659,A -85,B 0,C 180,E1 -19831.045,E2 -19831.045} C_VEL
LIN {X 0,Y 230.615,Z 679.192,A -85,B 0,C 180,E1 -19832.867,E2 -19832.867} C_VEL
LIN {X 0,Y 229.957,Z 680.924,A -85,B 0,C 180,E1 -19834.279,E2 -19834.279} C_VEL
LIN {X 0,Y 230,Z 681.438,A -85,B 0,C 180,E1 -19834.758,E2 -19834.758} C_VEL
LIN {X 0,Y 230.915,Z 685.719,A -85,B 0,C 180,E1 -19838.603,E2 -19838.603} C_VEL
LIN {X 0,Y 231.872,Z 690.763,A -85,B 0,C 180,E1 -19842.622,E2 -19842.622} C_VEL
LIN {X 0,Y 232.833,Z 696.025,A -85,B 0,C 180,E1 -19846.422,E2 -19846.422} C_VEL
LIN {X 0,Y 233.567,Z 701.204,A -85,B 0,C 180,E1 -19849.845,E2 -19849.845} C_VEL
LIN {X 0,Y 232.964,Z 704.311,A -85,B 0,C 180,E1 -19851.662,E2 -19851.662} C_VEL
LIN {X 0,Y 232.408,Z 706.24,A -85,B 0,C 180,E1 -19852.747,E2 -19852.747} C_VEL
LIN {X 0,Y 233.351,Z 710.282,A -85,B 0,C 180,E1 -19853.222,E2 -19853.222} C_VEL
LIN {X 0,Y 235.921,Z 720.748,A -85,B 0,C 180,E1 -19854.61,E2 -19854.61} C_VEL
LIN {X 0,Y 238.183,Z 734.428,A -85,B 0,C 180,E1 -19856.467,E2 -19856.467} C_VEL
LIN {X 0,Y 239.099,Z 747.293,A -85,B 0,C 180,E1 -19858.309,E2 -19858.309} C_VEL
LIN {X 0,Y 238.925,Z 759.489,A -85,B 0,C 180,E1 -19860.239,E2 -19860.239} C_VEL
LIN {X 0,Y 237.99,Z 770.093,A -85,B 0,C 180,E1 -19862.143,E2 -19862.143} C_VEL
LIN {X 0,Y 236.5,Z 779.221,A -85,B 0,C 180,E1 -19864.002,E2 -19864.002} C_VEL
LIN {X 0,Y 235.626,Z 784.685,A -85,B 0,C 180,E1 -19865.2,E2 -19865.2} C_VEL
LIN {X 0,Y 234.93,Z 795.168,A -85,B 0,C 180,E1 -19866.647,E2 -19866.647} C_VEL
LIN {X 0,Y 232.839,Z 806.499,A -85,B 0,C 180,E1 -19868.531,E2 -19868.531} C_VEL
LIN {X 0,Y 231.217,Z 815.755,A -85,B 0,C 180,E1 -19870.466,E2 -19870.466} C_VEL
LIN {X 0,Y 229.661,Z 824.209,A -85,B 0,C 180,E1 -19872.64,E2 -19872.64} C_VEL
LIN {X 0,Y 228.094,Z 832.426,A -85,B 0,C 180,E1 -19875.273,E2 -19875.273} C_VEL
LIN {X 0,Y 227.089,Z 838.018,A -85,B 0,C 180,E1 -19877.488,E2 -19877.488} C_VEL
LIN {X 0,Y 226.356,Z 843.461,A -85,B 0,C 180,E1 -19880.167,E2 -19880.167} C_VEL
LIN {X 0,Y 225.934,Z 847.675,A -85,B 0,C 180,E1 -19882.852,E2 -19882.852} C_VEL
LIN {X 0,Y 225.762,Z 850.231,A -85,B 0,C 180,E1 -19884.985,E2 -19884.985} C_VEL
LIN {X 0,Y 225.796,Z 852.86,A -85,B 0,C 180,E1 -19888.215,E2 -19888.215} C_VEL
LIN {X 0,Y 225.855,Z 853.727,A -85,B 0,C 180,E1 -19889.999,E2 -19889.999} C_VEL
LIN {X 0,Y 225.759,Z 854.146,A -85,B 0,C 180,E1 -19891.783,E2 -19891.783} C_VEL
LIN {X 0,Y 225.732,Z 853.755,A -85,B 0,C 180,E1 -19895.358,E2 -19895.358} C_VEL
LIN {X 0,Y 225.897,Z 852.981,A -85,B 0,C 180,E1 -19897.148,E2 -19897.148} C_VEL
LIN {X 0,Y 226.24,Z 851.778,A -85,B 0,C 180,E1 -19898.934,E2 -19898.934} C_VEL
LIN {X 0,Y 227.394,Z 848.133,A -85,B 0,C 180,E1 -19902.493,E2 -19902.493} C_VEL
LIN {X 0,Y 228.755,Z 844.238,A -85,B 0,C 180,E1 -19905.137,E2 -19905.137} C_VEL
LIN {X 0,Y 230.714,Z 839.256,A -85,B 0,C 180,E1 -19907.734,E2 -19907.734} C_VEL
LIN {X 0,Y 233.022,Z 833.168,A -85,B 0,C 180,E1 -19910.248,E2 -19910.248} C_VEL
LIN {X 0,Y 235.764,Z 825.395,A -85,B 0,C 180,E1 -19912.799,E2 -19912.799} C_VEL
LIN {X 0,Y 239.014,Z 815.935,A -85,B 0,C 180,E1 -19915.235,E2 -19915.235} C_VEL
LIN {X 0,Y 242.277,Z 806.239,A -85,B 0,C 180,E1 -19917.185,E2 -19917.185} C_VEL
LIN {X 0,Y 243.871,Z 800.593,A -85,B 0,C 180,E1 -19918.157,E2 -19918.157} C_VEL
LIN {X 0,Y 245.935,Z 789.407,A -85,B 0,C 180,E1 -19919.919,E2 -19919.919} C_VEL
LIN {X 0,Y 247.451,Z 777.902,A -85,B 0,C 180,E1 -19921.414,E2 -19921.414} C_VEL
LIN {X 0,Y 247.4,Z 766.557,A -85,B 0,C 180,E1 -19922.819,E2 -19922.819} C_VEL
LIN {X 0,Y 245.98,Z 754.019,A -85,B 0,C 180,E1 -19924.336,E2 -19924.336} C_VEL
LIN {X 0,Y 243.034,Z 740.975,A -85,B 0,C 180,E1 -19925.933,E2 -19925.933} C_VEL
LIN {X 0,Y 241.965,Z 737.083,A -85,B 0,C 180,E1 -19926.459,E2 -19926.459} C_VEL
LIN {X 0,Y 242.575,Z 727.753,A -85,B 0,C 180,E1 -19929.03,E2 -19929.03} C_VEL
LIN {X 0,Y 243.394,Z 719.435,A -85,B 0,C 180,E1 -19931.614,E2 -19931.614} C_VEL
LIN {X 0,Y 243.253,Z 717.095,A -85,B 0,C 180,E1 -19932.548,E2 -19932.548} C_VEL
LIN {X 0,Y 242.238,Z 710.546,A -85,B 0,C 180,E1 -19935.868,E2 -19935.868} C_VEL
LIN {X 0,Y 241.589,Z 703.736,A -85,B 0,C 180,E1 -19940.208,E2 -19940.208} C_VEL
LIN {X 0,Y 241.381,Z 701.353,A -85,B 0,C 180,E1 -19942.307,E2 -19942.307} C_VEL
LIN {X 0,Y 240.689,Z 699.624,A -85,B 0,C 180,E1 -19944.842,E2 -19944.842} C_VEL
LIN {X 0,Y 239.788,Z 698.395,A -85,B 0,C 180,E1 -19948.206,E2 -19948.206} C_VEL
LIN {X 0,Y 239.4,Z 698.007,A -85,B 0,C 180,E1 -19951.984,E2 -19951.984} C_VEL
LIN {X 0,Y 239.373,Z 698.105,A -85,B 0,C 180,E1 -19953.87,E2 -19953.87} C_VEL
LIN {X 0,Y 239.419,Z 699.271,A -85,B 0,C 180,E1 -19957.566,E2 -19957.566} C_VEL
LIN {X 0,Y 239.865,Z 701.279,A -85,B 0,C 180,E1 -19961.198,E2 -19961.198} C_VEL
LIN {X 0,Y 240.389,Z 704.018,A -85,B 0,C 180,E1 -19964.744,E2 -19964.744} C_VEL
LIN {X 0,Y 241.084,Z 707.424,A -85,B 0,C 180,E1 -19968.225,E2 -19968.225} C_VEL
LIN {X 0,Y 241.771,Z 711.454,A -85,B 0,C 180,E1 -19971.643,E2 -19971.643} C_VEL
LIN {X 0,Y 242.282,Z 717.444,A -85,B 0,C 180,E1 -19975.841,E2 -19975.841} C_VEL
LIN {X 0,Y 242.2,Z 721.59,A -85,B 0,C 180,E1 -19978.337,E2 -19978.337} C_VEL
LIN {X 0,Y 241.158,Z 726.515,A -85,B 0,C 180,E1 -19980.835,E2 -19980.835} C_VEL
LIN {X 0,Y 239.45,Z 733.045,A -85,B 0,C 180,E1 -19983.918,E2 -19983.918} C_VEL
LIN {X 0,Y 243.973,Z 747.358,A -85,B 0,C 180,E1 -19986.201,E2 -19986.201} C_VEL
LIN {X 0,Y 246.297,Z 758.602,A -85,B 0,C 180,E1 -19987.944,E2 -19987.944} C_VEL
LIN {X 0,Y 247.546,Z 770.306,A -85,B 0,C 180,E1 -19989.808,E2 -19989.808} C_VEL
LIN {X 0,Y 247.663,Z 780.177,A -85,B 0,C 180,E1 -19991.457,E2 -19991.457} C_VEL
LIN {X 0,Y 246.452,Z 785.808,A -85,B 0,C 180,E1 -19992.293,E2 -19992.293} C_VEL
LIN {X 0,Y 243.504,Z 795.996,A -85,B 0,C 180,E1 -19993.988,E2 -19993.988} C_VEL
LIN {X 0,Y 240.507,Z 805.127,A -85,B 0,C 180,E1 -19995.886,E2 -19995.886} C_VEL
LIN {X 0,Y 237.289,Z 814.236,A -85,B 0,C 180,E1 -19998.27,E2 -19998.27} C_VEL
LIN {X 0,Y 234.537,Z 821.383,A -85,B 0,C 180,E1 -20000.615,E2 -20000.615} C_VEL
LIN {X 0,Y 232.114,Z 827.561,A -85,B 0,C 180,E1 -20003.179,E2 -20003.179} C_VEL
LIN {X 0,Y 229.705,Z 833.169,A -85,B 0,C 180,E1 -20006.231,E2 -20006.231} C_VEL
LIN {X 0,Y 227.843,Z 837.577,A -85,B 0,C 180,E1 -20009.573,E2 -20009.573} C_VEL
LIN {X 0,Y 226.478,Z 840.462,A -85,B 0,C 180,E1 -20013.088,E2 -20013.088} C_VEL
LIN {X 0,Y 225.653,Z 841.727,A -85,B 0,C 180,E1 -20016.282,E2 -20016.282} C_VEL
LIN {X 0,Y 225.334,Z 841.813,A -85,B 0,C 180,E1 -20018.766,E2 -20018.766} C_VEL
LIN {X 0,Y 225.159,Z 841.032,A -85,B 0,C 180,E1 -20021.488,E2 -20021.488} C_VEL
LIN {X 0,Y 225.28,Z 839.359,A -85,B 0,C 180,E1 -20024.151,E2 -20024.151} C_VEL
LIN {X 0,Y 225.66,Z 836.814,A -85,B 0,C 180,E1 -20026.753,E2 -20026.753} C_VEL
LIN {X 0,Y 226.192,Z 833.427,A -85,B 0,C 180,E1 -20029.272,E2 -20029.272} C_VEL
LIN {X 0,Y 226.879,Z 829.175,A -85,B 0,C 180,E1 -20031.719,E2 -20031.719} C_VEL
LIN {X 0,Y 228.122,Z 822.641,A -85,B 0,C 180,E1 -20034.64,E2 -20034.64} C_VEL
LIN {X 0,Y 229.378,Z 815.905,A -85,B 0,C 180,E1 -20037.044,E2 -20037.044} C_VEL
LIN {X 0,Y 230.998,Z 807.902,A -85,B 0,C 180,E1 -20039.364,E2 -20039.364} C_VEL
LIN {X 0,Y 232.641,Z 799.549,A -85,B 0,C 180,E1 -20041.346,E2 -20041.346} C_VEL
LIN {X 0,Y 234.442,Z 789.554,A -85,B 0,C 180,E1 -20043.279,E2 -20043.279} C_VEL
LIN {X 0,Y 236.489,Z 777.105,A -85,B 0,C 180,E1 -20045.181,E2 -20045.181} C_VEL
LIN {X 0,Y 237.134,Z 771.078,A -85,B 0,C 180,E1 -20045.953,E2 -20045.953} C_VEL
LIN {X 0,Y 235.776,Z 758.075,A -85,B 0,C 180,E1 -20047.524,E2 -20047.524} C_VEL
LIN {X 0,Y 233.983,Z 745.186,A -85,B 0,C 180,E1 -20048.759,E2 -20048.759} C_VEL
LIN {X 0,Y 231.558,Z 731.376,A -85,B 0,C 180,E1 -20049.805,E2 -20049.805} C_VEL
LIN {X 0,Y 232.707,Z 721.997,A -85,B 0,C 180,E1 -20053.779,E2 -20053.779} C_VEL
LIN {X 0,Y 234.04,Z 711.401,A -85,B 0,C 180,E1 -20058.306,E2 -20058.306} C_VEL
LIN {X 0,Y 234.628,Z 706.039,A -85,B 0,C 180,E1 -20060.606,E2 -20060.606} C_VEL
LIN {X 0,Y 234.279,Z 700.585,A -85,B 0,C 180,E1 -20063.109,E2 -20063.109} C_VEL
LIN {X 0,Y 233.045,Z 693.464,A -85,B 0,C 180,E1 -20066.543,E2 -20066.543} C_VEL
LIN {X 0,Y 231.652,Z 684.863,A -85,B 0,C 180,E1 -20070.783,E2 -20070.783} C_VEL
LIN {X 0,Y 230.227,Z 679.668,A -85,B 0,C 180,E1 -20073.501,E2 -20073.501} C_VEL
LIN {X 0,Y 228.322,Z 672.043,A -85,B 0,C 180,E1 -20077.629,E2 -20077.629} C_VEL
LIN {X 0,Y 228.3,Z 672.213,A -85,B 0,C 180,E1 -20079.835,E2 -20079.835} C_VEL
LIN {X 0,Y 231.963,Z 682.917,A -85,B 0,C 180,E1 -20081.358,E2 -20081.358} C_VEL
LIN {X 0,Y 235.436,Z 693.659,A -85,B 0,C 180,E1 -20083.151,E2 -20083.151} C_VEL
LIN {X 0,Y 238.226,Z 704.335,A -85,B 0,C 180,E1 -20085.179,E2 -20085.179} C_VEL
LIN {X 0,Y 238.136,Z 706.79,A -85,B 0,C 180,E1 -20085.624,E2 -20085.624} C_VEL
LIN {X 0,Y 236.21,Z 717.961,A -85,B 0,C 180,E1 -20087.805,E2 -20087.805} C_VEL
LIN {X 0,Y 234.432,Z 727.542,A -85,B 0,C 180,E1 -20090.168,E2 -20090.168} C_VEL
LIN {X 0,Y 232.802,Z 735.595,A -85,B 0,C 180,E1 -20092.638,E2 -20092.638} C_VEL
LIN {X 0,Y 231.183,Z 743.421,A -85,B 0,C 180,E1 -20095.672,E2 -20095.672} C_VEL
LIN {X 0,Y 230.102,Z 748.926,A -85,B 0,C 180,E1 -20098.446,E2 -20098.446} C_VEL
LIN {X 0,Y 229.266,Z 753.405,A -85,B 0,C 180,E1 -20101.408,E2 -20101.408} C_VEL
LIN {X 0,Y 228.755,Z 756.234,A -85,B 0,C 180,E1 -20103.951,E2 -20103.951} C_VEL
LIN {X 0,Y 228.553,Z 758.43,A -85,B 0,C 180,E1 -20106.918,E2 -20106.918} C_VEL
LIN {X 0,Y 228.843,Z 759.556,A -85,B 0,C 180,E1 -20110.161,E2 -20110.161} C_VEL
LIN {X 0,Y 229.409,Z 759.484,A -85,B 0,C 180,E1 -20112.672,E2 -20112.672} C_VEL
LIN {X 0,Y 230.314,Z 758.506,A -85,B 0,C 180,E1 -20115.425,E2 -20115.425} C_VEL
LIN {X 0,Y 231.554,Z 756.581,A -85,B 0,C 180,E1 -20118.108,E2 -20118.108} C_VEL
LIN {X 0,Y 233.553,Z 752.708,A -85,B 0,C 180,E1 -20121.48,E2 -20121.48} C_VEL
LIN {X 0,Y 235.228,Z 749.026,A -85,B 0,C 180,E1 -20123.775,E2 -20123.775} C_VEL
LIN {X 0,Y 237.717,Z 743.162,A -85,B 0,C 180,E1 -20126.551,E2 -20126.551} C_VEL
LIN {X 0,Y 240.118,Z 736.863,A -85,B 0,C 180,E1 -20128.884,E2 -20128.884} C_VEL
LIN {X 0,Y 242.665,Z 729.396,A -85,B 0,C 180,E1 -20131.106,E2 -20131.106} C_VEL
LIN {X 0,Y 245.569,Z 720.006,A -85,B 0,C 180,E1 -20133.325,E2 -20133.325} C_VEL
LIN {X 0,Y 246.217,Z 717.566,A -85,B 0,C 180,E1 -20133.819,E2 -20133.819} C_VEL
LIN {X 0,Y 244.912,Z 709.939,A -85,B 0,C 180,E1 -20135.863,E2 -20135.863} C_VEL
LIN {X 0,Y 242.217,Z 700.854,A -85,B 0,C 180,E1 -20138.243,E2 -20138.243} C_VEL
LIN {X 0,Y 238.367,Z 691.224,A -85,B 0,C 180,E1 -20140.731,E2 -20140.731} C_VEL
LIN {X 0,Y 233.612,Z 681.924,A -85,B 0,C 180,E1 -20143.183,E2 -20143.183} C_VEL
LIN {X 0,Y 230.369,Z 676.496,A -85,B 0,C 180,E1 -20144.688,E2 -20144.688} C_VEL
LIN {X 0,Y 228.631,Z 674.109,A -85,B 0,C 180,E1 -20145.423,E2 -20145.423} C_VEL
LIN {X 0,Y 228.068,Z 672.073,A -85,B 0,C 180,E1 -20145.842,E2 -20145.842} C_VEL
LIN {X 0,Y 228.309,Z 672.041,A -85,B 0,C 180,E1 -20151.146,E2 -20151.146} C_VEL
LIN {X 0,Y 228.358,Z 672.027,A -85,B 0,C 180,E1 -20152.929,E2 -20152.929} C_VEL
LIN {X 0,Y 228.558,Z 672.01,A -85,B 0,C 180,E1 -20158.238,E2 -20158.238} C_VEL
LIN {X 0,Y 228.558,Z 672.003,A -85,B 0,C 180,E1 -20161.762,E2 -20161.762} C_VEL
LIN {X 0,Y 228.358,Z 672.04,A -85,B 0,C 180,E1 -20167.072,E2 -20167.072} C_VEL
LIN {X 0,Y 228.162,Z 672.062,A -85,B 0,C 180,E1 -20170.651,E2 -20170.651} C_VEL
LIN {X 0,Y 228.068,Z 672.072,A -85,B 0,C 180,E1 -20174.272,E2 -20174.272} C_VEL
LIN {X 0,Y 228.006,Z 672.081,A -85,B 0,C 180,E1 -20177.953,E2 -20177.953} C_VEL
LIN {X 0,Y 227.933,Z 672.087,A -85,B 0,C 180,E1 -20182.329,E2 -20182.329} C_VEL
LIN {X 0,Y 227.923,Z 672.14,A -85,B 0,C 180,E1 -20184.115,E2 -20184.115} C_VEL
LIN {X 0,Y 228.488,Z 674.683,A -85,B 0,C 180,E1 -20187.477,E2 -20187.477} C_VEL
LIN {X 0,Y 229.225,Z 678.118,A -85,B 0,C 180,E1 -20191.414,E2 -20191.414} C_VEL
LIN {X 0,Y 230,Z 681.438,A -85,B 0,C 180,E1 -20194.758,E2 -20194.758} C_VEL
LIN {X 0,Y 229.71,Z 683.156,A -85,B 0,C 180,E1 -20196.164,E2 -20196.164} C_VEL
LIN {X 0,Y 227.477,Z 686.555,A -85,B 0,C 180,E1 -20198.43,E2 -20198.43} C_VEL
LIN {X 0,Y 225.548,Z 689.428,A -85,B 0,C 180,E1 -20200.263,E2 -20200.263} C_VEL
LIN {X 0,Y 224.886,Z 691.457,A -85,B 0,C 180,E1 -20201.686,E2 -20201.686} C_VEL
LIN {X 0,Y 224.93,Z 692.081,A -85,B 0,C 180,E1 -20202.168,E2 -20202.168} C_VEL
LIN {X 0,Y 226.057,Z 698.361,A -85,B 0,C 180,E1 -20206.845,E2 -20206.845} C_VEL
LIN {X 0,Y 226.568,Z 702.041,A -85,B 0,C 180,E1 -20209.351,E2 -20209.351} C_VEL
LIN {X 0,Y 226.189,Z 704.886,A -85,B 0,C 180,E1 -20211.053,E2 -20211.053} C_VEL
LIN {X 0,Y 227.222,Z 709.171,A -85,B 0,C 180,E1 -20211.609,E2 -20211.609} C_VEL
LIN {X 0,Y 229.824,Z 719.748,A -85,B 0,C 180,E1 -20213.156,E2 -20213.156} C_VEL
LIN {X 0,Y 232.15,Z 734.094,A -85,B 0,C 180,E1 -20215.234,E2 -20215.234} C_VEL
LIN {X 0,Y 232.943,Z 746.382,A -85,B 0,C 180,E1 -20217.106,E2 -20217.106} C_VEL
LIN {X 0,Y 232.752,Z 758.483,A -85,B 0,C 180,E1 -20219.114,E2 -20219.114} C_VEL
LIN {X 0,Y 231.714,Z 769.585,A -85,B 0,C 180,E1 -20221.186,E2 -20221.186} C_VEL
LIN {X 0,Y 230.058,Z 779.094,A -85,B 0,C 180,E1 -20223.217,E2 -20223.217} C_VEL
LIN {X 0,Y 228.793,Z 785.368,A -85,B 0,C 180,E1 -20224.772,E2 -20224.772} C_VEL
LIN {X 0,Y 228.13,Z 794.983,A -85,B 0,C 180,E1 -20226.149,E2 -20226.149} C_VEL
LIN {X 0,Y 225.987,Z 806.308,A -85,B 0,C 180,E1 -20228.087,E2 -20228.087} C_VEL
LIN {X 0,Y 224.128,Z 816.274,A -85,B 0,C 180,E1 -20230.247,E2 -20230.247} C_VEL
LIN {X 0,Y 222.516,Z 824.751,A -85,B 0,C 180,E1 -20232.538,E2 -20232.538} C_VEL
LIN {X 0,Y 220.951,Z 832.844,A -85,B 0,C 180,E1 -20235.257,E2 -20235.257} C_VEL
LIN {X 0,Y 219.827,Z 839.335,A -85,B 0,C 180,E1 -20238.005,E2 -20238.005} C_VEL
LIN {X 0,Y 219.168,Z 844.444,A -85,B 0,C 180,E1 -20240.773,E2 -20240.773} C_VEL
LIN {X 0,Y 218.778,Z 848.355,A -85,B 0,C 180,E1 -20243.543,E2 -20243.543} C_VEL
LIN {X 0,Y 218.632,Z 851.191,A -85,B 0,C 180,E1 -20246.313,E2 -20246.313} C_VEL
LIN {X 0,Y 218.706,Z 852.508,A -85,B 0,C 180,E1 -20248.158,E2 -20248.158} C_VEL
LIN {X 0,Y 218.786,Z 853.416,A -85,B 0,C 180,E1 -20249.999,E2 -20249.999} C_VEL
LIN {X 0,Y 218.67,Z 853.91,A -85,B 0,C 180,E1 -20251.841,E2 -20251.841} C_VEL
LIN {X 0,Y 218.598,Z 853.841,A -85,B 0,C 180,E1 -20254.68,E2 -20254.68} C_VEL
LIN {X 0,Y 218.838,Z 852.886,A -85,B 0,C 180,E1 -20257.38,E2 -20257.38} C_VEL
LIN {X 0,Y 219.206,Z 851.764,A -85,B 0,C 180,E1 -20259.224,E2 -20259.224} C_VEL
LIN {X 0,Y 220.456,Z 848.228,A -85,B 0,C 180,E1 -20262.893,E2 -20262.893} C_VEL
LIN {X 0,Y 221.888,Z 844.458,A -85,B 0,C 180,E1 -20265.617,E2 -20265.617} C_VEL
LIN {X 0,Y 223.977,Z 839.595,A -85,B 0,C 180,E1 -20268.286,E2 -20268.286} C_VEL
LIN {X 0,Y 226.412,Z 833.523,A -85,B 0,C 180,E1 -20270.913,E2 -20270.913} C_VEL
LIN {X 0,Y 229.289,Z 826.065,A -85,B 0,C 180,E1 -20273.481,E2 -20273.481} C_VEL
LIN {X 0,Y 232.667,Z 816.858,A -85,B 0,C 180,E1 -20275.974,E2 -20275.974} C_VEL
LIN {X 0,Y 236.424,Z 806.426,A -85,B 0,C 180,E1 -20278.157,E2 -20278.157} C_VEL
LIN {X 0,Y 238.211,Z 799.684,A -85,B 0,C 180,E1 -20279.372,E2 -20279.372} C_VEL
LIN {X 0,Y 240.587,Z 787.83,A -85,B 0,C 180,E1 -20281.231,E2 -20281.231} C_VEL
LIN {X 0,Y 241.883,Z 777.764,A -85,B 0,C 180,E1 -20282.583,E2 -20282.583} C_VEL
LIN {X 0,Y 241.943,Z 767.357,A -85,B 0,C 180,E1 -20283.955,E2 -20283.955} C_VEL
LIN {X 0,Y 240.694,Z 755.314,A -85,B 0,C 180,E1 -20285.502,E2 -20285.502} C_VEL
LIN {X 0,Y 238.017,Z 742.7,A -85,B 0,C 180,E1 -20287.177,E2 -20287.177} C_VEL
LIN {X 0,Y 236.474,Z 736.79,A -85,B 0,C 180,E1 -20288.048,E2 -20288.048} C_VEL
LIN {X 0,Y 237.651,Z 725.161,A -85,B 0,C 180,E1 -20291.562,E2 -20291.562} C_VEL
LIN {X 0,Y 237.921,Z 721.728,A -85,B 0,C 180,E1 -20292.795,E2 -20292.795} C_VEL
LIN {X 0,Y 236.938,Z 714.788,A -85,B 0,C 180,E1 -20296.37,E2 -20296.37} C_VEL
LIN {X 0,Y 236.422,Z 708.3,A -85,B 0,C 180,E1 -20300.612,E2 -20300.612} C_VEL
LIN {X 0,Y 236.39,Z 707.39,A -85,B 0,C 180,E1 -20301.366,E2 -20301.366} C_VEL
LIN {X 0,Y 235.889,Z 705.412,A -85,B 0,C 180,E1 -20303.553,E2 -20303.553} C_VEL
LIN {X 0,Y 235.377,Z 704.246,A -85,B 0,C 180,E1 -20305.437,E2 -20305.437} C_VEL
LIN {X 0,Y 234.311,Z 702.866,A -85,B 0,C 180,E1 -20310.437,E2 -20310.437} C_VEL
LIN {X 0,Y 234.05,Z 702.918,A -85,B 0,C 180,E1 -20314.265,E2 -20314.265} C_VEL
LIN {X 0,Y 234.091,Z 704.389,A -85,B 0,C 180,E1 -20318.54,E2 -20318.54} C_VEL
LIN {X 0,Y 234.46,Z 706.673,A -85,B 0,C 180,E1 -20322.557,E2 -20322.557} C_VEL
LIN {X 0,Y 234.95,Z 709.619,A -85,B 0,C 180,E1 -20326.154,E2 -20326.154} C_VEL
LIN {X 0,Y 235.581,Z 713.425,A -85,B 0,C 180,E1 -20329.883,E2 -20329.883} C_VEL
LIN {X 0,Y 235.808,Z 716.426,A -85,B 0,C 180,E1 -20332.292,E2 -20332.292} C_VEL
LIN {X 0,Y 236.203,Z 721.134,A -85,B 0,C 180,E1 -20335.734,E2 -20335.734} C_VEL
LIN {X 0,Y 235.913,Z 725.331,A -85,B 0,C 180,E1 -20338.293,E2 -20338.293} C_VEL
LIN {X 0,Y 234.653,Z 730.339,A -85,B 0,C 180,E1 -20340.858,E2 -20340.858} C_VEL
LIN {X 0,Y 233.815,Z 733.22,A -85,B 0,C 180,E1 -20342.261,E2 -20342.261} C_VEL
LIN {X 0,Y 237.941,Z 746.421,A -85,B 0,C 180,E1 -20344.542,E2 -20344.542} C_VEL
LIN {X 0,Y 240.291,Z 757.046,A -85,B 0,C 180,E1 -20346.334,E2 -20346.334} C_VEL
LIN {X 0,Y 241.644,Z 767.279,A -85,B 0,C 180,E1 -20348.049,E2 -20348.049} C_VEL
LIN {X 0,Y 241.941,Z 777.484,A -85,B 0,C 180,E1 -20349.805,E2 -20349.805} C_VEL
LIN {X 0,Y 241.789,Z 782.332,A -85,B 0,C 180,E1 -20350.678,E2 -20350.678} C_VEL
LIN {X 0,Y 238.56,Z 793.852,A -85,B 0,C 180,E1 -20352.533,E2 -20352.533} C_VEL
LIN {X 0,Y 235.253,Z 803.601,A -85,B 0,C 180,E1 -20354.489,E2 -20354.489} C_VEL
LIN {X 0,Y 231.975,Z 812.439,A -85,B 0,C 180,E1 -20356.727,E2 -20356.727} C_VEL
LIN {X 0,Y 228.613,Z 820.744,A -85,B 0,C 180,E1 -20359.427,E2 -20359.427} C_VEL
LIN {X 0,Y 225.569,Z 827.938,A -85,B 0,C 180,E1 -20362.437,E2 -20362.437} C_VEL
LIN {X 0,Y 223.225,Z 833.036,A -85,B 0,C 180,E1 -20365.258,E2 -20365.258} C_VEL
LIN {X 0,Y 221.27,Z 837.255,A -85,B 0,C 180,E1 -20368.452,E2 -20368.452} C_VEL
LIN {X 0,Y 220.271,Z 839.39,A -85,B 0,C 180,E1 -20370.697,E2 -20370.697} C_VEL
LIN {X 0,Y 219.221,Z 841.191,A -85,B 0,C 180,E1 -20373.539,E2 -20373.539} C_VEL
LIN {X 0,Y 218.527,Z 842.038,A -85,B 0,C 180,E1 -20376.487,E2 -20376.487} C_VEL
LIN {X 0,Y 218.132,Z 841.669,A -85,B 0,C 180,E1 -20380.119,E2 -20380.119} C_VEL
LIN {X 0,Y 218.07,Z 840.536,A -85,B 0,C 180,E1 -20382.593,E2 -20382.593} C_VEL
LIN {X 0,Y 218.268,Z 838.645,A -85,B 0,C 180,E1 -20385.103,E2 -20385.103} C_VEL
LIN {X 0,Y 218.737,Z 835.894,A -85,B 0,C 180,E1 -20387.645,E2 -20387.645} C_VEL
LIN {X 0,Y 219.481,Z 831.099,A -85,B 0,C 180,E1 -20390.859,E2 -20390.859} C_VEL
LIN {X 0,Y 220.726,Z 824.774,A -85,B 0,C 180,E1 -20394.026,E2 -20394.026} C_VEL
LIN {X 0,Y 221.922,Z 818.356,A -85,B 0,C 180,E1 -20396.558,E2 -20396.558} C_VEL
LIN {X 0,Y 223.775,Z 809.544,A -85,B 0,C 180,E1 -20399.314,E2 -20399.314} C_VEL
LIN {X 0,Y 225.604,Z 800.415,A -85,B 0,C 180,E1 -20401.603,E2 -20401.603} C_VEL
LIN {X 0,Y 227.629,Z 789.721,A -85,B 0,C 180,E1 -20403.748,E2 -20403.748} C_VEL
LIN {X 0,Y 229.741,Z 777.248,A -85,B 0,C 180,E1 -20405.705,E2 -20405.705} C_VEL
